LIN {X 0,Y 411.23,Z 342.072,A -85,B 0,C 180,E1 -10466.382,E2 -10466.382} C_VEL
LIN {X 0,Y 411.203,Z 342.077,A -85,B 0,C 180,E1 -10469.713,E2 -10469.713} C_VEL
LIN {X 0,Y 411.199,Z 342.079,A -85,B 0,C 180,E1 -10473.157,E2 -10473.157} C_VEL
LIN {X 0,Y 411.189,Z 342.079,A -85,B 0,C 180,E1 -10476.555,E2 -10476.555} C_VEL
LIN {X 0,Y 411.209,Z 342.075,A -85,B 0,C 180,E1 -10479.73,E2 -10479.73} C_VEL
LIN {X 0,Y 411.172,Z 342.082,A -85,B 0,C 180,E1 -10483.135,E2 -10483.135} C_VEL
LIN {X 0,Y 411.168,Z 342.08,A -85,B 0,C 180,E1 -10485.882,E2 -10485.882} C_VEL
LIN {X 0,Y 411.161,Z 342.084,A -85,B 0,C 180,E1 -10488.773,E2 -10488.773} C_VEL
LIN {X 0,Y 411.202,Z 342.076,A -85,B 0,C 180,E1 -10492.029,E2 -10492.029} C_VEL
LIN {X 0,Y 412.209,Z 347.522,A -85,B 0,C 180,E1 -10494.924,E2 -10494.924} C_VEL
LIN {X 0,Y 412.634,Z 351.681,A -85,B 0,C 180,E1 -10496.975,E2 -10496.975} C_VEL
LIN {X 0,Y 412.275,Z 356.532,A -85,B 0,C 180,E1 -10499.244,E2 -10499.244} C_VEL
LIN {X 0,Y 411.689,Z 363.91,A -85,B 0,C 180,E1 -10502.586,E2 -10502.586} C_VEL
LIN {X 0,Y 411.232,Z 371.157,A -85,B 0,C 180,E1 -10505.787,E2 -10505.787} C_VEL
LIN {X 0,Y 410.777,Z 379.693,A -85,B 0,C 180,E1 -10509.469,E2 -10509.469} C_VEL
LIN {X 0,Y 410.455,Z 388.245,A -85,B 0,C 180,E1 -10513.079,E2 -10513.079} C_VEL
LIN {X 0,Y 410.22,Z 395.922,A -85,B 0,C 180,E1 -10516.264,E2 -10516.264} C_VEL
LIN {X 0,Y 411.645,Z 408.983,A -85,B 0,C 180,E1 -10516.82,E2 -10516.82} C_VEL
LIN {X 0,Y 412.334,Z 417.705,A -85,B 0,C 180,E1 -10517.325,E2 -10517.325} C_VEL
LIN {X 0,Y 412.266,Z 426.417,A -85,B 0,C 180,E1 -10517.948,E2 -10517.948} C_VEL
LIN {X 0,Y 411.784,Z 434.733,A -85,B 0,C 180,E1 -10518.682,E2 -10518.682} C_VEL
LIN {X 0,Y 411.383,Z 442.624,A -85,B 0,C 180,E1 -10519.543,E2 -10519.543} C_VEL
LIN {X 0,Y 410.961,Z 449.152,A -85,B 0,C 180,E1 -10520.403,E2 -10520.403} C_VEL
LIN {X 0,Y 410.635,Z 455.373,A -85,B 0,C 180,E1 -10521.389,E2 -10521.389} C_VEL
LIN {X 0,Y 410.389,Z 460.538,A -85,B 0,C 180,E1 -10522.375,E2 -10522.375} C_VEL
LIN {X 0,Y 410.192,Z 464.991,A -85,B 0,C 180,E1 -10523.399,E2 -10523.399} C_VEL
LIN {X 0,Y 410.072,Z 469.17,A -85,B 0,C 180,E1 -10524.592,E2 -10524.592} C_VEL
LIN {X 0,Y 410.022,Z 471.91,A -85,B 0,C 180,E1 -10525.578,E2 -10525.578} C_VEL
LIN {X 0,Y 410.004,Z 474.894,A -85,B 0,C 180,E1 -10527.054,E2 -10527.054} C_VEL
LIN {X 0,Y 410.022,Z 476.211,A -85,B 0,C 180,E1 -10528.037,E2 -10528.037} C_VEL
LIN {X 0,Y 409.977,Z 477.041,A -85,B 0,C 180,E1 -10529.019,E2 -10529.019} C_VEL
LIN {X 0,Y 409.971,Z 477.337,A -85,B 0,C 180,E1 -10530.001,E2 -10530.001} C_VEL
LIN {X 0,Y 409.977,Z 477.054,A -85,B 0,C 180,E1 -10530.983,E2 -10530.983} C_VEL
LIN {X 0,Y 410.021,Z 476.298,A -85,B 0,C 180,E1 -10531.966,E2 -10531.966} C_VEL
LIN {X 0,Y 409.989,Z 475.058,A -85,B 0,C 180,E1 -10532.949,E2 -10532.949} C_VEL
LIN {X 0,Y 410.022,Z 472.138,A -85,B 0,C 180,E1 -10534.425,E2 -10534.425} C_VEL
LIN {X 0,Y 410.073,Z 469.497,A -85,B 0,C 180,E1 -10535.41,E2 -10535.41} C_VEL
LIN {X 0,Y 410.211,Z 465.349,A -85,B 0,C 180,E1 -10536.622,E2 -10536.622} C_VEL
LIN {X 0,Y 410.407,Z 461.101,A -85,B 0,C 180,E1 -10537.628,E2 -10537.628} C_VEL
LIN {X 0,Y 410.667,Z 456.097,A -85,B 0,C 180,E1 -10538.613,E2 -10538.613} C_VEL
LIN {X 0,Y 411.002,Z 450.082,A -85,B 0,C 180,E1 -10539.598,E2 -10539.598} C_VEL
LIN {X 0,Y 411.478,Z 442.783,A -85,B 0,C 180,E1 -10540.581,E2 -10540.581} C_VEL
LIN {X 0,Y 411.898,Z 435.006,A -85,B 0,C 180,E1 -10541.442,E2 -10541.442} C_VEL
LIN {X 0,Y 412.411,Z 426.855,A -85,B 0,C 180,E1 -10542.175,E2 -10542.175} C_VEL
LIN {X 0,Y 412.692,Z 420.277,A -85,B 0,C 180,E1 -10542.667,E2 -10542.667} C_VEL
LIN {X 0,Y 412.229,Z 412.315,A -85,B 0,C 180,E1 -10543.177,E2 -10543.177} C_VEL
LIN {X 0,Y 411.234,Z 402.961,A -85,B 0,C 180,E1 -10543.655,E2 -10543.655} C_VEL
LIN {X 0,Y 410.211,Z 395.094,A -85,B 0,C 180,E1 -10544.006,E2 -10544.006} C_VEL
LIN {X 0,Y 410.526,Z 386.814,A -85,B 0,C 180,E1 -10547.434,E2 -10547.434} C_VEL
LIN {X 0,Y 410.847,Z 378.285,A -85,B 0,C 180,E1 -10551.054,E2 -10551.054} C_VEL
LIN {X 0,Y 411.287,Z 370.025,A -85,B 0,C 180,E1 -10554.664,E2 -10554.664} C_VEL
LIN {X 0,Y 411.817,Z 362.717,A -85,B 0,C 180,E1 -10557.991,E2 -10557.991} C_VEL
LIN {X 0,Y 412.393,Z 356.864,A -85,B 0,C 180,E1 -10560.749,E2 -10560.749} C_VEL
LIN {X 0,Y 412.717,Z 352.266,A -85,B 0,C 180,E1 -10563.02,E2 -10563.02} C_VEL
LIN {X 0,Y 412.292,Z 348.349,A -85,B 0,C 180,E1 -10565.093,E2 -10565.093} C_VEL
LIN {X 0,Y 411.234,Z 342.076,A -85,B 0,C 180,E1 -10568.7,E2 -10568.7} C_VEL
LIN {X 0,Y 411.184,Z 342.088,A -85,B 0,C 180,E1 -10571.806,E2 -10571.806} C_VEL
LIN {X 0,Y 411.183,Z 342.084,A -85,B 0,C 180,E1 -10575.51,E2 -10575.51} C_VEL
LIN {X 0,Y 411.17,Z 342.083,A -85,B 0,C 180,E1 -10578.772,E2 -10578.772} C_VEL
LIN {X 0,Y 411.197,Z 342.079,A -85,B 0,C 180,E1 -10582.026,E2 -10582.026} C_VEL
LIN {X 0,Y 411.212,Z 342.078,A -85,B 0,C 180,E1 -10585.666,E2 -10585.666} C_VEL
LIN {X 0,Y 411.197,Z 342.079,A -85,B 0,C 180,E1 -10589.152,E2 -10589.152} C_VEL
LIN {X 0,Y 411.266,Z 342.069,A -85,B 0,C 180,E1 -10592.522,E2 -10592.522} C_VEL
LIN {X 0,Y 411.234,Z 342.074,A -85,B 0,C 180,E1 -10595.784,E2 -10595.784} C_VEL
LIN {X 0,Y 411.204,Z 342.079,A -85,B 0,C 180,E1 -10598.966,E2 -10598.966} C_VEL
LIN {X 0,Y 411.258,Z 342.071,A -85,B 0,C 180,E1 -10602.084,E2 -10602.084} C_VEL
LIN {X 0,Y 411.267,Z 342.07,A -85,B 0,C 180,E1 -10605.147,E2 -10605.147} C_VEL
LIN {X 0,Y 411.29,Z 342.068,A -85,B 0,C 180,E1 -10608.167,E2 -10608.167} C_VEL
LIN {X 0,Y 411.325,Z 342.062,A -85,B 0,C 180,E1 -10611.153,E2 -10611.153} C_VEL
LIN {X 0,Y 411.448,Z 342.048,A -85,B 0,C 180,E1 -10614.117,E2 -10614.117} C_VEL
LIN {X 0,Y 411.515,Z 342.037,A -85,B 0,C 180,E1 -10618.042,E2 -10618.042} C_VEL
LIN {X 0,Y 411.646,Z 342.024,A -85,B 0,C 180,E1 -10619.999,E2 -10619.999} C_VEL
LIN {X 0,Y 411.461,Z 342.045,A -85,B 0,C 180,E1 -10622.936,E2 -10622.936} C_VEL
LIN {X 0,Y 411.438,Z 342.048,A -85,B 0,C 180,E1 -10626.627,E2 -10626.627} C_VEL
LIN {X 0,Y 411.323,Z 342.062,A -85,B 0,C 180,E1 -10628.845,E2 -10628.845} C_VEL
LIN {X 0,Y 411.287,Z 342.069,A -85,B 0,C 180,E1 -10631.832,E2 -10631.832} C_VEL
LIN {X 0,Y 411.261,Z 342.074,A -85,B 0,C 180,E1 -10634.851,E2 -10634.851} C_VEL
LIN {X 0,Y 411.086,Z 342.096,A -85,B 0,C 180,E1 -10637.921,E2 -10637.921} C_VEL
LIN {X 0,Y 410.952,Z 342.111,A -85,B 0,C 180,E1 -10638.96,E2 -10638.96} C_VEL
LIN {X 0,Y 410.855,Z 342.735,A -85,B 0,C 180,E1 -10640.005,E2 -10640.005} C_VEL
LIN {X 0,Y 410.697,Z 346.204,A -85,B 0,C 180,E1 -10643.176,E2 -10643.176} C_VEL
LIN {X 0,Y 410.524,Z 349.853,A -85,B 0,C 180,E1 -10646.429,E2 -10646.429} C_VEL
LIN {X 0,Y 410.4,Z 353.677,A -85,B 0,C 180,E1 -10649.775,E2 -10649.775} C_VEL
LIN {X 0,Y 410.282,Z 357.723,A -85,B 0,C 180,E1 -10653.239,E2 -10653.239} C_VEL
LIN {X 0,Y 410.198,Z 361.362,A -85,B 0,C 180,E1 -10656.158,E2 -10656.158} C_VEL
LIN {X 0,Y 412.433,Z 371.958,A -85,B 0,C 180,E1 -10656.694,E2 -10656.694} C_VEL
LIN {X 0,Y 413.573,Z 378.962,A -85,B 0,C 180,E1 -10657.125,E2 -10657.125} C_VEL
LIN {X 0,Y 413.1,Z 389.049,A -85,B 0,C 180,E1 -10657.844,E2 -10657.844} C_VEL
LIN {X 0,Y 412.623,Z 397.601,A -85,B 0,C 180,E1 -10658.62,E2 -10658.62} C_VEL
LIN {X 0,Y 412.151,Z 405.235,A -85,B 0,C 180,E1 -10659.474,E2 -10659.474} C_VEL
LIN {X 0,Y 411.705,Z 412.313,A -85,B 0,C 180,E1 -10660.44,E2 -10660.44} C_VEL
LIN {X 0,Y 411.181,Z 420.303,A -85,B 0,C 180,E1 -10661.803,E2 -10661.803} C_VEL
LIN {X 0,Y 410.704,Z 426.486,A -85,B 0,C 180,E1 -10663.193,E2 -10663.193} C_VEL
LIN {X 0,Y 410.422,Z 431.277,A -85,B 0,C 180,E1 -10664.592,E2 -10664.592} C_VEL
LIN {X 0,Y 410.205,Z 434.884,A -85,B 0,C 180,E1 -10666.018,E2 -10666.018} C_VEL
LIN {X 0,Y 409.984,Z 437.361,A -85,B 0,C 180,E1 -10667.484,E2 -10667.484} C_VEL
LIN {X 0,Y 409.867,Z 438.729,A -85,B 0,C 180,E1 -10669.337,E2 -10669.337} C_VEL
LIN {X 0,Y 409.875,Z 438.684,A -85,B 0,C 180,E1 -10670.621,E2 -10670.621} C_VEL
LIN {X 0,Y 409.906,Z 437.633,A -85,B 0,C 180,E1 -10672.061,E2 -10672.061} C_VEL
LIN {X 0,Y 410.115,Z 435.241,A -85,B 0,C 180,E1 -10673.649,E2 -10673.649} C_VEL
LIN {X 0,Y 410.267,Z 432.368,A -85,B 0,C 180,E1 -10674.875,E2 -10674.875} C_VEL
LIN {X 0,Y 410.556,Z 427.036,A -85,B 0,C 180,E1 -10676.49,E2 -10676.49} C_VEL
LIN {X 0,Y 410.9,Z 421.655,A -85,B 0,C 180,E1 -10677.737,E2 -10677.737} C_VEL
LIN {X 0,Y 411.219,Z 416.518,A -85,B 0,C 180,E1 -10678.705,E2 -10678.705} C_VEL
LIN {X 0,Y 411.616,Z 409.786,A -85,B 0,C 180,E1 -10679.755,E2 -10679.755} C_VEL
LIN {X 0,Y 411.963,Z 402.423,A -85,B 0,C 180,E1 -10680.698,E2 -10680.698} C_VEL
LIN {X 0,Y 412.553,Z 392.414,A -85,B 0,C 180,E1 -10681.717,E2 -10681.717} C_VEL
LIN {X 0,Y 412.981,Z 382.762,A -85,B 0,C 180,E1 -10682.465,E2 -10682.465} C_VEL
LIN {X 0,Y 413.008,Z 376.343,A -85,B 0,C 180,E1 -10682.88,E2 -10682.88} C_VEL
LIN {X 0,Y 411.176,Z 365.69,A -85,B 0,C 180,E1 -10683.452,E2 -10683.452} C_VEL
LIN {X 0,Y 410.147,Z 360.352,A -85,B 0,C 180,E1 -10683.714,E2 -10683.714} C_VEL
LIN {X 0,Y 410.174,Z 356.533,A -85,B 0,C 180,E1 -10686.79,E2 -10686.79} C_VEL
LIN {X 0,Y 410.288,Z 352.106,A -85,B 0,C 180,E1 -10690.406,E2 -10690.406} C_VEL
LIN {X 0,Y 410.442,Z 348.369,A -85,B 0,C 180,E1 -10693.508,E2 -10693.508} C_VEL
LIN {X 0,Y 410.61,Z 343.854,A -85,B 0,C 180,E1 -10697.313,E2 -10697.313} C_VEL
LIN {X 0,Y 410.673,Z 342.882,A -85,B 0,C 180,E1 -10698.148,E2 -10698.148} C_VEL
LIN {X 0,Y 410.706,Z 342.14,A -85,B 0,C 180,E1 -10699.149,E2 -10699.149} C_VEL
LIN {X 0,Y 411.303,Z 342.067,A -85,B 0,C 180,E1 -10702.319,E2 -10702.319} C_VEL
LIN {X 0,Y 411.449,Z 342.048,A -85,B 0,C 180,E1 -10704.116,E2 -10704.116} C_VEL
LIN {X 0,Y 411.504,Z 342.041,A -85,B 0,C 180,E1 -10708.041,E2 -10708.041} C_VEL
LIN {X 0,Y 411.631,Z 342.025,A -85,B 0,C 180,E1 -10709.999,E2 -10709.999} C_VEL
LIN {X 0,Y 411.457,Z 342.044,A -85,B 0,C 180,E1 -10712.936,E2 -10712.936} C_VEL
LIN {X 0,Y 411.482,Z 342.045,A -85,B 0,C 180,E1 -10715.881,E2 -10715.881} C_VEL
LIN {X 0,Y 411.444,Z 342.045,A -85,B 0,C 180,E1 -10717.13,E2 -10717.13} C_VEL
LIN {X 0,Y 410.763,Z 342.134,A -85,B 0,C 180,E1 -10717.947,E2 -10717.947} C_VEL
LIN {X 0,Y 407.846,Z 342.494,A -85,B 0,C 180,E1 -10719.272,E2 -10719.272} C_VEL
LIN {X 0,Y 405.379,Z 342.803,A -85,B 0,C 180,E1 -10720.343,E2 -10720.343} C_VEL
LIN {X 0,Y 404.323,Z 342.933,A -85,B 0,C 180,E1 -10721.172,E2 -10721.172} C_VEL
LIN {X 0,Y 404.239,Z 342.942,A -85,B 0,C 180,E1 -10721.452,E2 -10721.452} C_VEL
LIN {X 0,Y 404.204,Z 342.95,A -85,B 0,C 180,E1 -10724.087,E2 -10724.087} C_VEL
LIN {X 0,Y 404.19,Z 342.951,A -85,B 0,C 180,E1 -10727.192,E2 -10727.192} C_VEL
LIN {X 0,Y 404.15,Z 342.954,A -85,B 0,C 180,E1 -10730.351,E2 -10730.351} C_VEL
LIN {X 0,Y 404.156,Z 342.957,A -85,B 0,C 180,E1 -10733.574,E2 -10733.574} C_VEL
LIN {X 0,Y 404.17,Z 342.954,A -85,B 0,C 180,E1 -10735.766,E2 -10735.766} C_VEL
LIN {X 0,Y 404.184,Z 342.951,A -85,B 0,C 180,E1 -10737.999,E2 -10737.999} C_VEL
LIN {X 0,Y 404.129,Z 342.959,A -85,B 0,C 180,E1 -10741.558,E2 -10741.558} C_VEL
LIN {X 0,Y 404.171,Z 342.954,A -85,B 0,C 180,E1 -10745.016,E2 -10745.016} C_VEL
LIN {X 0,Y 404.149,Z 342.956,A -85,B 0,C 180,E1 -10748.755,E2 -10748.755} C_VEL
LIN {X 0,Y 404.177,Z 342.953,A -85,B 0,C 180,E1 -10751.61,E2 -10751.61} C_VEL
LIN {X 0,Y 404.184,Z 342.951,A -85,B 0,C 180,E1 -10754.53,E2 -10754.53} C_VEL
LIN {X 0,Y 404.192,Z 342.951,A -85,B 0,C 180,E1 -10757.305,E2 -10757.305} C_VEL
LIN {X 0,Y 404.154,Z 342.953,A -85,B 0,C 180,E1 -10759.955,E2 -10759.955} C_VEL
LIN {X 0,Y 404.126,Z 342.959,A -85,B 0,C 180,E1 -10763.124,E2 -10763.124} C_VEL
LIN {X 0,Y 404.13,Z 342.957,A -85,B 0,C 180,E1 -10766.188,E2 -10766.188} C_VEL
LIN {X 0,Y 404.14,Z 342.954,A -85,B 0,C 180,E1 -10769.716,E2 -10769.716} C_VEL
LIN {X 0,Y 404.181,Z 342.951,A -85,B 0,C 180,E1 -10773.123,E2 -10773.123} C_VEL
LIN {X 0,Y 404.169,Z 342.955,A -85,B 0,C 180,E1 -10776.427,E2 -10776.427} C_VEL
LIN {X 0,Y 404.213,Z 342.946,A -85,B 0,C 180,E1 -10779.861,E2 -10779.861} C_VEL
LIN {X 0,Y 404.205,Z 342.948,A -85,B 0,C 180,E1 -10782.992,E2 -10782.992} C_VEL
LIN {X 0,Y 404.253,Z 342.943,A -85,B 0,C 180,E1 -10786.789,E2 -10786.789} C_VEL
LIN {X 0,Y 404.258,Z 342.944,A -85,B 0,C 180,E1 -10789.989,E2 -10789.989} C_VEL
LIN {X 0,Y 404.4,Z 342.923,A -85,B 0,C 180,E1 -10793.014,E2 -10793.014} C_VEL
LIN {X 0,Y 404.273,Z 342.938,A -85,B 0,C 180,E1 -10795.015,E2 -10795.015} C_VEL
LIN {X 0,Y 404.471,Z 342.917,A -85,B 0,C 180,E1 -10798.009,E2 -10798.009} C_VEL
LIN {X 0,Y 404.6,Z 342.901,A -85,B 0,C 180,E1 -10800.001,E2 -10800.001} C_VEL
LIN {X 0,Y 404.415,Z 342.921,A -85,B 0,C 180,E1 -10802.989,E2 -10802.989} C_VEL
LIN {X 0,Y 404.401,Z 342.923,A -85,B 0,C 180,E1 -10806.988,E2 -10806.988} C_VEL
LIN {X 0,Y 404.261,Z 342.943,A -85,B 0,C 180,E1 -10810.013,E2 -10810.013} C_VEL
LIN {X 0,Y 404.256,Z 342.943,A -85,B 0,C 180,E1 -10813.213,E2 -10813.213} C_VEL
LIN {X 0,Y 404.206,Z 342.949,A -85,B 0,C 180,E1 -10817.008,E2 -10817.008} C_VEL
LIN {X 0,Y 404.155,Z 342.953,A -85,B 0,C 180,E1 -10820.353,E2 -10820.353} C_VEL
LIN {X 0,Y 404.161,Z 342.956,A -85,B 0,C 180,E1 -10823.576,E2 -10823.576} C_VEL
LIN {X 0,Y 404.175,Z 342.953,A -85,B 0,C 180,E1 -10825.768,E2 -10825.768} C_VEL
LIN {X 0,Y 404.19,Z 342.949,A -85,B 0,C 180,E1 -10828.001,E2 -10828.001} C_VEL
LIN {X 0,Y 404.135,Z 342.958,A -85,B 0,C 180,E1 -10831.56,E2 -10831.56} C_VEL
LIN {X 0,Y 404.178,Z 342.954,A -85,B 0,C 180,E1 -10835.017,E2 -10835.017} C_VEL
LIN {X 0,Y 404.151,Z 342.957,A -85,B 0,C 180,E1 -10838.758,E2 -10838.758} C_VEL
LIN {X 0,Y 404.118,Z 342.959,A -85,B 0,C 180,E1 -10841.601,E2 -10841.601} C_VEL
LIN {X 0,Y 404.144,Z 342.957,A -85,B 0,C 180,E1 -10844.524,E2 -10844.524} C_VEL
LIN {X 0,Y 404.134,Z 342.958,A -85,B 0,C 180,E1 -10847.298,E2 -10847.298} C_VEL
LIN {X 0,Y 404.164,Z 342.954,A -85,B 0,C 180,E1 -10849.957,E2 -10849.957} C_VEL
LIN {X 0,Y 404.201,Z 343.069,A -85,B 0,C 180,E1 -10851.965,E2 -10851.965} C_VEL
LIN {X 0,Y 405.47,Z 350.234,A -85,B 0,C 180,E1 -10855.717,E2 -10855.717} C_VEL
LIN {X 0,Y 405.604,Z 353.875,A -85,B 0,C 180,E1 -10857.512,E2 -10857.512} C_VEL
LIN {X 0,Y 404.93,Z 361.148,A -85,B 0,C 180,E1 -10860.926,E2 -10860.926} C_VEL
LIN {X 0,Y 404.403,Z 368.438,A -85,B 0,C 180,E1 -10864.25,E2 -10864.25} C_VEL
LIN {X 0,Y 403.922,Z 375.737,A -85,B 0,C 180,E1 -10867.495,E2 -10867.495} C_VEL
LIN {X 0,Y 403.561,Z 383.066,A -85,B 0,C 180,E1 -10870.679,E2 -10870.679} C_VEL
LIN {X 0,Y 403.312,Z 390.352,A -85,B 0,C 180,E1 -10873.812,E2 -10873.812} C_VEL
LIN {X 0,Y 403.117,Z 395.66,A -85,B 0,C 180,E1 -10876.058,E2 -10876.058} C_VEL
LIN {X 0,Y 404.579,Z 408.507,A -85,B 0,C 180,E1 -10876.603,E2 -10876.603} C_VEL
LIN {X 0,Y 405.268,Z 417.013,A -85,B 0,C 180,E1 -10877.1,E2 -10877.1} C_VEL
LIN {X 0,Y 405.302,Z 425.811,A -85,B 0,C 180,E1 -10877.737,E2 -10877.737} C_VEL
LIN {X 0,Y 404.817,Z 434.179,A -85,B 0,C 180,E1 -10878.485,E2 -10878.485} C_VEL
LIN {X 0,Y 404.396,Z 442.112,A -85,B 0,C 180,E1 -10879.361,E2 -10879.361} C_VEL
LIN {X 0,Y 403.94,Z 448.67,A -85,B 0,C 180,E1 -10880.235,E2 -10880.235} C_VEL
LIN {X 0,Y 403.601,Z 454.919,A -85,B 0,C 180,E1 -10881.237,E2 -10881.237} C_VEL
LIN {X 0,Y 403.327,Z 460.107,A -85,B 0,C 180,E1 -10882.24,E2 -10882.24} C_VEL
LIN {X 0,Y 403.116,Z 464.859,A -85,B 0,C 180,E1 -10883.356,E2 -10883.356} C_VEL
LIN {X 0,Y 402.972,Z 468.776,A -85,B 0,C 180,E1 -10884.497,E2 -10884.497} C_VEL
LIN {X 0,Y 402.952,Z 471.534,A -85,B 0,C 180,E1 -10885.5,E2 -10885.5} C_VEL
LIN {X 0,Y 402.904,Z 474.529,A -85,B 0,C 180,E1 -10887.002,E2 -10887.002} C_VEL
LIN {X 0,Y 402.951,Z 475.861,A -85,B 0,C 180,E1 -10888.002,E2 -10888.002} C_VEL
LIN {X 0,Y 402.902,Z 476.702,A -85,B 0,C 180,E1 -10889.002,E2 -10889.002} C_VEL
LIN {X 0,Y 402.894,Z 477,A -85,B 0,C 180,E1 -10890.001,E2 -10890.001} C_VEL
LIN {X 0,Y 402.902,Z 476.726,A -85,B 0,C 180,E1 -10891.001,E2 -10891.001} C_VEL
LIN {X 0,Y 402.95,Z 475.982,A -85,B 0,C 180,E1 -10892,E2 -10892} C_VEL
LIN {X 0,Y 402.888,Z 474.753,A -85,B 0,C 180,E1 -10893.001,E2 -10893.001} C_VEL
LIN {X 0,Y 402.952,Z 471.848,A -85,B 0,C 180,E1 -10894.503,E2 -10894.503} C_VEL
LIN {X 0,Y 402.971,Z 469.219,A -85,B 0,C 180,E1 -10895.506,E2 -10895.506} C_VEL
LIN {X 0,Y 403.137,Z 465.344,A -85,B 0,C 180,E1 -10896.672,E2 -10896.672} C_VEL
LIN {X 0,Y 403.359,Z 460.853,A -85,B 0,C 180,E1 -10897.762,E2 -10897.762} C_VEL
LIN {X 0,Y 403.617,Z 455.866,A -85,B 0,C 180,E1 -10898.765,E2 -10898.765} C_VEL
LIN {X 0,Y 403.988,Z 449.872,A -85,B 0,C 180,E1 -10899.767,E2 -10899.767} C_VEL
LIN {X 0,Y 404.5,Z 442.599,A -85,B 0,C 180,E1 -10900.766,E2 -10900.766} C_VEL
LIN {X 0,Y 404.947,Z 434.855,A -85,B 0,C 180,E1 -10901.641,E2 -10901.641} C_VEL
LIN {X 0,Y 405.48,Z 426.747,A -85,B 0,C 180,E1 -10902.387,E2 -10902.387} C_VEL
LIN {X 0,Y 405.686,Z 420.228,A -85,B 0,C 180,E1 -10902.889,E2 -10902.889} C_VEL
LIN {X 0,Y 405.115,Z 411.093,A -85,B 0,C 180,E1 -10903.481,E2 -10903.481} C_VEL
LIN {X 0,Y 404.054,Z 401.482,A -85,B 0,C 180,E1 -10903.97,E2 -10903.97} C_VEL
LIN {X 0,Y 403.148,Z 394.806,A -85,B 0,C 180,E1 -10904.256,E2 -10904.256} C_VEL
LIN {X 0,Y 403.457,Z 386.563,A -85,B 0,C 180,E1 -10907.75,E2 -10907.75} C_VEL
LIN {X 0,Y 403.81,Z 378.069,A -85,B 0,C 180,E1 -10911.439,E2 -10911.439} C_VEL
LIN {X 0,Y 404.239,Z 370.846,A -85,B 0,C 180,E1 -10914.663,E2 -10914.663} C_VEL
LIN {X 0,Y 404.786,Z 363.737,A -85,B 0,C 180,E1 -10917.956,E2 -10917.956} C_VEL
LIN {X 0,Y 405.441,Z 356.773,A -85,B 0,C 180,E1 -10921.335,E2 -10921.335} C_VEL
LIN {X 0,Y 405.723,Z 353.363,A -85,B 0,C 180,E1 -10923.07,E2 -10923.07} C_VEL
LIN {X 0,Y 405.359,Z 349.966,A -85,B 0,C 180,E1 -10924.901,E2 -10924.901} C_VEL
LIN {X 0,Y 404.324,Z 343.717,A -85,B 0,C 180,E1 -10928.537,E2 -10928.537} C_VEL
LIN {X 0,Y 404.185,Z 342.955,A -85,B 0,C 180,E1 -10929.075,E2 -10929.075} C_VEL
LIN {X 0,Y 404.16,Z 342.963,A -85,B 0,C 180,E1 -10933.084,E2 -10933.084} C_VEL
LIN {X 0,Y 404.155,Z 342.959,A -85,B 0,C 180,E1 -10935.926,E2 -10935.926} C_VEL
LIN {X 0,Y 404.125,Z 342.961,A -85,B 0,C 180,E1 -10938.635,E2 -10938.635} C_VEL
LIN {X 0,Y 404.155,Z 342.956,A -85,B 0,C 180,E1 -10941.493,E2 -10941.493} C_VEL
LIN {X 0,Y 404.191,Z 342.952,A -85,B 0,C 180,E1 -10944.984,E2 -10944.984} C_VEL
LIN {X 0,Y 404.149,Z 342.957,A -85,B 0,C 180,E1 -10948.554,E2 -10948.554} C_VEL
LIN {X 0,Y 404.203,Z 342.95,A -85,B 0,C 180,E1 -10952,E2 -10952} C_VEL
LIN {X 0,Y 404.185,Z 342.953,A -85,B 0,C 180,E1 -10955.334,E2 -10955.334} C_VEL
LIN {X 0,Y 404.146,Z 342.957,A -85,B 0,C 180,E1 -10958.58,E2 -10958.58} C_VEL
LIN {X 0,Y 404.216,Z 342.947,A -85,B 0,C 180,E1 -10961.761,E2 -10961.761} C_VEL
LIN {X 0,Y 404.213,Z 342.95,A -85,B 0,C 180,E1 -10964.881,E2 -10964.881} C_VEL
LIN {X 0,Y 404.262,Z 342.942,A -85,B 0,C 180,E1 -10967.958,E2 -10967.958} C_VEL
LIN {X 0,Y 404.272,Z 342.941,A -85,B 0,C 180,E1 -10970.998,E2 -10970.998} C_VEL
LIN {X 0,Y 404.398,Z 342.926,A -85,B 0,C 180,E1 -10974.014,E2 -10974.014} C_VEL
LIN {X 0,Y 404.484,Z 342.913,A -85,B 0,C 180,E1 -10978.008,E2 -10978.008} C_VEL
LIN {X 0,Y 404.615,Z 342.9,A -85,B 0,C 180,E1 -10979.999,E2 -10979.999} C_VEL
LIN {X 0,Y 404.419,Z 342.922,A -85,B 0,C 180,E1 -10982.987,E2 -10982.987} C_VEL
LIN {X 0,Y 404.387,Z 342.926,A -85,B 0,C 180,E1 -10986.625,E2 -10986.625} C_VEL
LIN {X 0,Y 404.261,Z 342.943,A -85,B 0,C 180,E1 -10990.011,E2 -10990.011} C_VEL
LIN {X 0,Y 404.271,Z 342.945,A -85,B 0,C 180,E1 -10993.21,E2 -10993.21} C_VEL
LIN {X 0,Y 404.204,Z 342.954,A -85,B 0,C 180,E1 -10996.151,E2 -10996.151} C_VEL
LIN {X 0,Y 403.844,Z 342.997,A -85,B 0,C 180,E1 -10999.307,E2 -10999.307} C_VEL
LIN {X 0,Y 403.694,Z 346.515,A -85,B 0,C 180,E1 -11002.676,E2 -11002.676} C_VEL
LIN {X 0,Y 403.5,Z 350.007,A -85,B 0,C 180,E1 -11005.812,E2 -11005.812} C_VEL
LIN {X 0,Y 403.359,Z 354.027,A -85,B 0,C 180,E1 -11009.402,E2 -11009.402} C_VEL
LIN {X 0,Y 403.229,Z 357.821,A -85,B 0,C 180,E1 -11012.703,E2 -11012.703} C_VEL
LIN {X 0,Y 403.109,Z 361.529,A -85,B 0,C 180,E1 -11015.869,E2 -11015.869} C_VEL
LIN {X 0,Y 405.442,Z 372.434,A -85,B 0,C 180,E1 -11016.443,E2 -11016.443} C_VEL
LIN {X 0,Y 406.673,Z 379.898,A -85,B 0,C 180,E1 -11016.923,E2 -11016.923} C_VEL
LIN {X 0,Y 406.245,Z 388.915,A -85,B 0,C 180,E1 -11017.574,E2 -11017.574} C_VEL
LIN {X 0,Y 405.797,Z 396.48,A -85,B 0,C 180,E1 -11018.252,E2 -11018.252} C_VEL
LIN {X 0,Y 405.348,Z 403.228,A -85,B 0,C 180,E1 -11018.979,E2 -11018.979} C_VEL
LIN {X 0,Y 404.874,Z 410.673,A -85,B 0,C 180,E1 -11019.959,E2 -11019.959} C_VEL
LIN {X 0,Y 404.441,Z 417.301,A -85,B 0,C 180,E1 -11021.026,E2 -11021.026} C_VEL
LIN {X 0,Y 404.106,Z 421.562,A -85,B 0,C 180,E1 -11021.836,E2 -11021.836} C_VEL
LIN {X 0,Y 403.686,Z 426.671,A -85,B 0,C 180,E1 -11023.012,E2 -11023.012} C_VEL
LIN {X 0,Y 403.436,Z 430.702,A -85,B 0,C 180,E1 -11024.17,E2 -11024.17} C_VEL
LIN {X 0,Y 403.183,Z 434.518,A -85,B 0,C 180,E1 -11025.615,E2 -11025.615} C_VEL
LIN {X 0,Y 402.936,Z 437.29,A -85,B 0,C 180,E1 -11027.137,E2 -11027.137} C_VEL
LIN {X 0,Y 402.828,Z 438.814,A -85,B 0,C 180,E1 -11028.606,E2 -11028.606} C_VEL
LIN {X 0,Y 402.761,Z 439.179,A -85,B 0,C 180,E1 -11030.153,E2 -11030.153} C_VEL
LIN {X 0,Y 402.799,Z 438.304,A -85,B 0,C 180,E1 -11031.733,E2 -11031.733} C_VEL
LIN {X 0,Y 402.847,Z 437.676,A -85,B 0,C 180,E1 -11032.366,E2 -11032.366} C_VEL
LIN {X 0,Y 403.025,Z 435.668,A -85,B 0,C 180,E1 -11033.636,E2 -11033.636} C_VEL
LIN {X 0,Y 403.194,Z 432.506,A -85,B 0,C 180,E1 -11035.007,E2 -11035.007} C_VEL
LIN {X 0,Y 403.461,Z 427.845,A -85,B 0,C 180,E1 -11036.454,E2 -11036.454} C_VEL
LIN {X 0,Y 403.802,Z 422.952,A -85,B 0,C 180,E1 -11037.641,E2 -11037.641} C_VEL
LIN {X 0,Y 404.054,Z 418.484,A -85,B 0,C 180,E1 -11038.545,E2 -11038.545} C_VEL
LIN {X 0,Y 404.537,Z 411.162,A -85,B 0,C 180,E1 -11039.746,E2 -11039.746} C_VEL
LIN {X 0,Y 404.925,Z 404.086,A -85,B 0,C 180,E1 -11040.694,E2 -11040.694} C_VEL
LIN {X 0,Y 405.364,Z 396.557,A -85,B 0,C 180,E1 -11041.524,E2 -11041.524} C_VEL
LIN {X 0,Y 405.858,Z 386.656,A -85,B 0,C 180,E1 -11042.404,E2 -11042.404} C_VEL
LIN {X 0,Y 406.177,Z 378.2,A -85,B 0,C 180,E1 -11042.985,E2 -11042.985} C_VEL
LIN {X 0,Y 404.21,Z 366.469,A -85,B 0,C 180,E1 -11043.645,E2 -11043.645} C_VEL
LIN {X 0,Y 403.075,Z 360.681,A -85,B 0,C 180,E1 -11043.913,E2 -11043.913} C_VEL
LIN {X 0,Y 403.098,Z 357.669,A -85,B 0,C 180,E1 -11046.358,E2 -11046.358} C_VEL
LIN {X 0,Y 403.213,Z 352.945,A -85,B 0,C 180,E1 -11050.252,E2 -11050.252} C_VEL
LIN {X 0,Y 403.383,Z 348.711,A -85,B 0,C 180,E1 -11053.812,E2 -11053.812} C_VEL
LIN {X 0,Y 403.541,Z 344.704,A -85,B 0,C 180,E1 -11057.228,E2 -11057.228} C_VEL
LIN {X 0,Y 403.628,Z 343.023,A -85,B 0,C 180,E1 -11058.957,E2 -11058.957} C_VEL
LIN {X 0,Y 404.246,Z 342.946,A -85,B 0,C 180,E1 -11062.283,E2 -11062.283} C_VEL
LIN {X 0,Y 404.391,Z 342.927,A -85,B 0,C 180,E1 -11064.013,E2 -11064.013} C_VEL
LIN {X 0,Y 404.473,Z 342.917,A -85,B 0,C 180,E1 -11068.007,E2 -11068.007} C_VEL
LIN {X 0,Y 404.601,Z 342.901,A -85,B 0,C 180,E1 -11069.999,E2 -11069.999} C_VEL
LIN {X 0,Y 404.414,Z 342.921,A -85,B 0,C 180,E1 -11072.987,E2 -11072.987} C_VEL
LIN {X 0,Y 404.428,Z 342.923,A -85,B 0,C 180,E1 -11075.984,E2 -11075.984} C_VEL
LIN {X 0,Y 404.411,Z 342.925,A -85,B 0,C 180,E1 -11077.99,E2 -11077.99} C_VEL
LIN {X 0,Y 404.239,Z 342.942,A -85,B 0,C 180,E1 -11081.452,E2 -11081.452} C_VEL
LIN {X 0,Y 403.574,Z 343.028,A -85,B 0,C 180,E1 -11082.284,E2 -11082.284} C_VEL
LIN {X 0,Y 400.709,Z 343.385,A -85,B 0,C 180,E1 -11083.636,E2 -11083.636} C_VEL
LIN {X 0,Y 398.279,Z 343.687,A -85,B 0,C 180,E1 -11084.728,E2 -11084.728} C_VEL
LIN {X 0,Y 397.232,Z 343.819,A -85,B 0,C 180,E1 -11085.573,E2 -11085.573} C_VEL
LIN {X 0,Y 397.145,Z 343.826,A -85,B 0,C 180,E1 -11085.859,E2 -11085.859} C_VEL
LIN {X 0,Y 397.149,Z 343.826,A -85,B 0,C 180,E1 -11088.573,E2 -11088.573} C_VEL
LIN {X 0,Y 397.083,Z 343.837,A -85,B 0,C 180,E1 -11091.818,E2 -11091.818} C_VEL
LIN {X 0,Y 397.143,Z 343.828,A -85,B 0,C 180,E1 -11095.131,E2 -11095.131} C_VEL
LIN {X 0,Y 397.149,Z 343.828,A -85,B 0,C 180,E1 -11097.776,E2 -11097.776} C_VEL
LIN {X 0,Y 397.07,Z 343.837,A -85,B 0,C 180,E1 -11100.881,E2 -11100.881} C_VEL
LIN {X 0,Y 397.111,Z 343.83,A -85,B 0,C 180,E1 -11104.493,E2 -11104.493} C_VEL
LIN {X 0,Y 397.096,Z 343.832,A -85,B 0,C 180,E1 -11108.274,E2 -11108.274} C_VEL
LIN {X 0,Y 397.141,Z 343.827,A -85,B 0,C 180,E1 -11111.993,E2 -11111.993} C_VEL
LIN {X 0,Y 397.135,Z 343.831,A -85,B 0,C 180,E1 -11115.06,E2 -11115.06} C_VEL
LIN {X 0,Y 397.141,Z 343.827,A -85,B 0,C 180,E1 -11118.007,E2 -11118.007} C_VEL
LIN {X 0,Y 397.096,Z 343.833,A -85,B 0,C 180,E1 -11121.726,E2 -11121.726} C_VEL
LIN {X 0,Y 397.111,Z 343.831,A -85,B 0,C 180,E1 -11125.507,E2 -11125.507} C_VEL
LIN {X 0,Y 397.072,Z 343.837,A -85,B 0,C 180,E1 -11129.119,E2 -11129.119} C_VEL
LIN {X 0,Y 397.18,Z 343.826,A -85,B 0,C 180,E1 -11132.61,E2 -11132.61} C_VEL
LIN {X 0,Y 397.126,Z 343.83,A -85,B 0,C 180,E1 -11135.983,E2 -11135.983} C_VEL
LIN {X 0,Y 397.143,Z 343.826,A -85,B 0,C 180,E1 -11139.274,E2 -11139.274} C_VEL
LIN {X 0,Y 397.17,Z 343.825,A -85,B 0,C 180,E1 -11142.844,E2 -11142.844} C_VEL
LIN {X 0,Y 397.17,Z 343.824,A -85,B 0,C 180,E1 -11145.658,E2 -11145.658} C_VEL
LIN {X 0,Y 397.197,Z 343.82,A -85,B 0,C 180,E1 -11148.778,E2 -11148.778} C_VEL
LIN {X 0,Y 397.382,Z 343.8,A -85,B 0,C 180,E1 -11152.042,E2 -11152.042} C_VEL
LIN {X 0,Y 397.244,Z 343.813,A -85,B 0,C 180,E1 -11154.926,E2 -11154.926} C_VEL
LIN {X 0,Y 397.44,Z 343.793,A -85,B 0,C 180,E1 -11157.974,E2 -11157.974} C_VEL
LIN {X 0,Y 397.569,Z 343.777,A -85,B 0,C 180,E1 -11160.001,E2 -11160.001} C_VEL
LIN {X 0,Y 397.373,Z 343.798,A -85,B 0,C 180,E1 -11163.042,E2 -11163.042} C_VEL
LIN {X 0,Y 397.353,Z 343.801,A -85,B 0,C 180,E1 -11167.113,E2 -11167.113} C_VEL
LIN {X 0,Y 397.219,Z 343.819,A -85,B 0,C 180,E1 -11170.192,E2 -11170.192} C_VEL
LIN {X 0,Y 397.217,Z 343.821,A -85,B 0,C 180,E1 -11173.322,E2 -11173.322} C_VEL
LIN {X 0,Y 397.172,Z 343.825,A -85,B 0,C 180,E1 -11177.156,E2 -11177.156} C_VEL
LIN {X 0,Y 397.094,Z 343.833,A -85,B 0,C 180,E1 -11180.731,E2 -11180.731} C_VEL
LIN {X 0,Y 397.124,Z 343.829,A -85,B 0,C 180,E1 -11184.02,E2 -11184.02} C_VEL
LIN {X 0,Y 397.187,Z 343.825,A -85,B 0,C 180,E1 -11187.391,E2 -11187.391} C_VEL
LIN {X 0,Y 397.077,Z 343.837,A -85,B 0,C 180,E1 -11190.883,E2 -11190.883} C_VEL
LIN {X 0,Y 397.119,Z 343.83,A -85,B 0,C 180,E1 -11194.495,E2 -11194.495} C_VEL
LIN {X 0,Y 397.099,Z 343.832,A -85,B 0,C 180,E1 -11198.276,E2 -11198.276} C_VEL
LIN {X 0,Y 397.083,Z 343.838,A -85,B 0,C 180,E1 -11200.91,E2 -11200.91} C_VEL
LIN {X 0,Y 397.098,Z 343.832,A -85,B 0,C 180,E1 -11203.65,E2 -11203.65} C_VEL
LIN {X 0,Y 397.1,Z 343.834,A -85,B 0,C 180,E1 -11206.522,E2 -11206.522} C_VEL
LIN {X 0,Y 397.111,Z 343.833,A -85,B 0,C 180,E1 -11210.425,E2 -11210.425} C_VEL
LIN {X 0,Y 397.142,Z 343.893,A -85,B 0,C 180,E1 -11211.732,E2 -11211.732} C_VEL
LIN {X 0,Y 398.238,Z 349.993,A -85,B 0,C 180,E1 -11215.004,E2 -11215.004} C_VEL
LIN {X 0,Y 398.604,Z 353.628,A -85,B 0,C 180,E1 -11216.869,E2 -11216.869} C_VEL
LIN {X 0,Y 398.097,Z 359.888,A -85,B 0,C 180,E1 -11219.889,E2 -11219.889} C_VEL
LIN {X 0,Y 397.507,Z 366.949,A -85,B 0,C 180,E1 -11223.204,E2 -11223.204} C_VEL
LIN {X 0,Y 397,Z 374.243,A -85,B 0,C 180,E1 -11226.53,E2 -11226.53} C_VEL
LIN {X 0,Y 396.576,Z 381.837,A -85,B 0,C 180,E1 -11229.927,E2 -11229.927} C_VEL
LIN {X 0,Y 396.245,Z 390.015,A -85,B 0,C 180,E1 -11233.515,E2 -11233.515} C_VEL
LIN {X 0,Y 396.049,Z 395.374,A -85,B 0,C 180,E1 -11235.833,E2 -11235.833} C_VEL
LIN {X 0,Y 397.489,Z 407.945,A -85,B 0,C 180,E1 -11236.373,E2 -11236.373} C_VEL
LIN {X 0,Y 398.291,Z 418.186,A -85,B 0,C 180,E1 -11237,E2 -11237} C_VEL
LIN {X 0,Y 398.341,Z 425.189,A -85,B 0,C 180,E1 -11237.52,E2 -11237.52} C_VEL
LIN {X 0,Y 397.82,Z 433.607,A -85,B 0,C 180,E1 -11238.28,E2 -11238.28} C_VEL
LIN {X 0,Y 397.373,Z 441.579,A -85,B 0,C 180,E1 -11239.17,E2 -11239.17} C_VEL
LIN {X 0,Y 396.93,Z 448.173,A -85,B 0,C 180,E1 -11240.061,E2 -11240.061} C_VEL
LIN {X 0,Y 396.572,Z 454.45,A -85,B 0,C 180,E1 -11241.081,E2 -11241.081} C_VEL
LIN {X 0,Y 396.273,Z 459.662,A -85,B 0,C 180,E1 -11242.101,E2 -11242.101} C_VEL
LIN {X 0,Y 396.022,Z 464.968,A -85,B 0,C 180,E1 -11243.378,E2 -11243.378} C_VEL
LIN {X 0,Y 395.874,Z 468.37,A -85,B 0,C 180,E1 -11244.398,E2 -11244.398} C_VEL
LIN {X 0,Y 395.881,Z 471.148,A -85,B 0,C 180,E1 -11245.419,E2 -11245.419} C_VEL
LIN {X 0,Y 395.805,Z 474.159,A -85,B 0,C 180,E1 -11246.948,E2 -11246.948} C_VEL
LIN {X 0,Y 395.881,Z 475.507,A -85,B 0,C 180,E1 -11247.967,E2 -11247.967} C_VEL
LIN {X 0,Y 395.83,Z 476.362,A -85,B 0,C 180,E1 -11248.984,E2 -11248.984} C_VEL
LIN {X 0,Y 395.819,Z 476.66,A -85,B 0,C 180,E1 -11250.001,E2 -11250.001} C_VEL
LIN {X 0,Y 395.83,Z 476.398,A -85,B 0,C 180,E1 -11251.019,E2 -11251.019} C_VEL
LIN {X 0,Y 395.861,Z 475.667,A -85,B 0,C 180,E1 -11252.036,E2 -11252.036} C_VEL
LIN {X 0,Y 395.788,Z 474.45,A -85,B 0,C 180,E1 -11253.055,E2 -11253.055} C_VEL
LIN {X 0,Y 395.882,Z 471.558,A -85,B 0,C 180,E1 -11254.583,E2 -11254.583} C_VEL
LIN {X 0,Y 395.912,Z 467.389,A -85,B 0,C 180,E1 -11256.115,E2 -11256.115} C_VEL
LIN {X 0,Y 396.242,Z 461.776,A -85,B 0,C 180,E1 -11257.646,E2 -11257.646} C_VEL
LIN {X 0,Y 396.582,Z 455.636,A -85,B 0,C 180,E1 -11258.922,E2 -11258.922} C_VEL
LIN {X 0,Y 396.98,Z 449.662,A -85,B 0,C 180,E1 -11259.941,E2 -11259.941} C_VEL
LIN {X 0,Y 397.515,Z 442.414,A -85,B 0,C 180,E1 -11260.957,E2 -11260.957} C_VEL
LIN {X 0,Y 398.009,Z 434.711,A -85,B 0,C 180,E1 -11261.847,E2 -11261.847} C_VEL
LIN {X 0,Y 398.563,Z 426.664,A -85,B 0,C 180,E1 -11262.605,E2 -11262.605} C_VEL
LIN {X 0,Y 398.703,Z 420.229,A -85,B 0,C 180,E1 -11263.119,E2 -11263.119} C_VEL
LIN {X 0,Y 398.205,Z 411.649,A -85,B 0,C 180,E1 -11263.697,E2 -11263.697} C_VEL
LIN {X 0,Y 397.142,Z 401.996,A -85,B 0,C 180,E1 -11264.214,E2 -11264.214} C_VEL
LIN {X 0,Y 396.099,Z 394.458,A -85,B 0,C 180,E1 -11264.548,E2 -11264.548} C_VEL
LIN {X 0,Y 396.405,Z 386.315,A -85,B 0,C 180,E1 -11268.076,E2 -11268.076} C_VEL
LIN {X 0,Y 396.786,Z 377.873,A -85,B 0,C 180,E1 -11271.838,E2 -11271.838} C_VEL
LIN {X 0,Y 397.331,Z 369.773,A -85,B 0,C 180,E1 -11275.565,E2 -11275.565} C_VEL
LIN {X 0,Y 397.936,Z 362.483,A -85,B 0,C 180,E1 -11279.058,E2 -11279.058} C_VEL
LIN {X 0,Y 398.607,Z 356.235,A -85,B 0,C 180,E1 -11282.187,E2 -11282.187} C_VEL
LIN {X 0,Y 398.632,Z 352.754,A -85,B 0,C 180,E1 -11284.042,E2 -11284.042} C_VEL
LIN {X 0,Y 397.682,Z 347.085,A -85,B 0,C 180,E1 -11287.32,E2 -11287.32} C_VEL
LIN {X 0,Y 397.177,Z 343.83,A -85,B 0,C 180,E1 -11289.373,E2 -11289.373} C_VEL
LIN {X 0,Y 397.109,Z 343.84,A -85,B 0,C 180,E1 -11293.479,E2 -11293.479} C_VEL
LIN {X 0,Y 397.109,Z 343.837,A -85,B 0,C 180,E1 -11296.521,E2 -11296.521} C_VEL
LIN {X 0,Y 397.119,Z 343.832,A -85,B 0,C 180,E1 -11300.423,E2 -11300.423} C_VEL
LIN {X 0,Y 397.115,Z 343.833,A -85,B 0,C 180,E1 -11304.265,E2 -11304.265} C_VEL
LIN {X 0,Y 397.122,Z 343.832,A -85,B 0,C 180,E1 -11306.727,E2 -11306.727} C_VEL
LIN {X 0,Y 397.132,Z 343.831,A -85,B 0,C 180,E1 -11310.296,E2 -11310.296} C_VEL
LIN {X 0,Y 397.202,Z 343.822,A -85,B 0,C 180,E1 -11312.61,E2 -11312.61} C_VEL
LIN {X 0,Y 397.14,Z 343.829,A -85,B 0,C 180,E1 -11315.981,E2 -11315.981} C_VEL
LIN {X 0,Y 397.146,Z 343.829,A -85,B 0,C 180,E1 -11319.704,E2 -11319.704} C_VEL
LIN {X 0,Y 397.189,Z 343.822,A -85,B 0,C 180,E1 -11322.844,E2 -11322.844} C_VEL
LIN {X 0,Y 397.236,Z 343.817,A -85,B 0,C 180,E1 -11326.702,E2 -11326.702} C_VEL
LIN {X 0,Y 397.223,Z 343.819,A -85,B 0,C 180,E1 -11329.808,E2 -11329.808} C_VEL
LIN {X 0,Y 397.324,Z 343.808,A -85,B 0,C 180,E1 -11332.887,E2 -11332.887} C_VEL
LIN {X 0,Y 397.25,Z 343.816,A -85,B 0,C 180,E1 -11334.924,E2 -11334.924} C_VEL
LIN {X 0,Y 397.453,Z 343.789,A -85,B 0,C 180,E1 -11337.972,E2 -11337.972} C_VEL
LIN {X 0,Y 397.584,Z 343.776,A -85,B 0,C 180,E1 -11339.999,E2 -11339.999} C_VEL
LIN {X 0,Y 397.379,Z 343.799,A -85,B 0,C 180,E1 -11343.04,E2 -11343.04} C_VEL
LIN {X 0,Y 397.338,Z 343.804,A -85,B 0,C 180,E1 -11346.621,E2 -11346.621} C_VEL
LIN {X 0,Y 397.24,Z 343.817,A -85,B 0,C 180,E1 -11349.161,E2 -11349.161} C_VEL
LIN {X 0,Y 397.223,Z 343.82,A -85,B 0,C 180,E1 -11352.257,E2 -11352.257} C_VEL
LIN {X 0,Y 397.175,Z 343.831,A -85,B 0,C 180,E1 -11355.391,E2 -11355.391} C_VEL
LIN {X 0,Y 397.019,Z 343.849,A -85,B 0,C 180,E1 -11357.512,E2 -11357.512} C_VEL
LIN {X 0,Y 396.787,Z 344.26,A -85,B 0,C 180,E1 -11359.665,E2 -11359.665} C_VEL
LIN {X 0,Y 396.632,Z 347.727,A -85,B 0,C 180,E1 -11362.942,E2 -11362.942} C_VEL
LIN {X 0,Y 396.434,Z 351.373,A -85,B 0,C 180,E1 -11366.307,E2 -11366.307} C_VEL
LIN {X 0,Y 396.279,Z 355.213,A -85,B 0,C 180,E1 -11369.772,E2 -11369.772} C_VEL
LIN {X 0,Y 396.164,Z 359.474,A -85,B 0,C 180,E1 -11373.509,E2 -11373.509} C_VEL
LIN {X 0,Y 396.053,Z 361.857,A -85,B 0,C 180,E1 -11375.581,E2 -11375.581} C_VEL
LIN {X 0,Y 398.539,Z 373.427,A -85,B 0,C 180,E1 -11376.209,E2 -11376.209} C_VEL
LIN {X 0,Y 399.798,Z 380.783,A -85,B 0,C 180,E1 -11376.702,E2 -11376.702} C_VEL
LIN {X 0,Y 399.346,Z 389.697,A -85,B 0,C 180,E1 -11377.366,E2 -11377.366} C_VEL
LIN {X 0,Y 398.876,Z 397.332,A -85,B 0,C 180,E1 -11378.072,E2 -11378.072} C_VEL
LIN {X 0,Y 398.407,Z 403.665,A -85,B 0,C 180,E1 -11378.771,E2 -11378.771} C_VEL
LIN {X 0,Y 397.939,Z 410.823,A -85,B 0,C 180,E1 -11379.728,E2 -11379.728} C_VEL
LIN {X 0,Y 397.448,Z 417.745,A -85,B 0,C 180,E1 -11380.862,E2 -11380.862} C_VEL
LIN {X 0,Y 396.998,Z 423.259,A -85,B 0,C 180,E1 -11381.966,E2 -11381.966} C_VEL
LIN {X 0,Y 396.627,Z 427.528,A -85,B 0,C 180,E1 -11383.005,E2 -11383.005} C_VEL
LIN {X 0,Y 396.351,Z 431.697,A -85,B 0,C 180,E1 -11384.267,E2 -11384.267} C_VEL
LIN {X 0,Y 396.178,Z 434.154,A -85,B 0,C 180,E1 -11385.199,E2 -11385.199} C_VEL
LIN {X 0,Y 395.906,Z 437.065,A -85,B 0,C 180,E1 -11386.702,E2 -11386.702} C_VEL
LIN {X 0,Y 395.763,Z 438.86,A -85,B 0,C 180,E1 -11388.229,E2 -11388.229} C_VEL
LIN {X 0,Y 395.698,Z 439.549,A -85,B 0,C 180,E1 -11389.791,E2 -11389.791} C_VEL
LIN {X 0,Y 395.727,Z 438.805,A -85,B 0,C 180,E1 -11391.566,E2 -11391.566} C_VEL
LIN {X 0,Y 395.842,Z 437.052,A -85,B 0,C 180,E1 -11393.028,E2 -11393.028} C_VEL
LIN {X 0,Y 396.022,Z 434.988,A -85,B 0,C 180,E1 -11394.151,E2 -11394.151} C_VEL
LIN {X 0,Y 396.274,Z 430.165,A -85,B 0,C 180,E1 -11395.965,E2 -11395.965} C_VEL
LIN {X 0,Y 396.687,Z 424.024,A -85,B 0,C 180,E1 -11397.592,E2 -11397.592} C_VEL
LIN {X 0,Y 397.092,Z 417.971,A -85,B 0,C 180,E1 -11398.822,E2 -11398.822} C_VEL
LIN {X 0,Y 397.507,Z 411.739,A -85,B 0,C 180,E1 -11399.856,E2 -11399.856} C_VEL
LIN {X 0,Y 397.91,Z 404.918,A -85,B 0,C 180,E1 -11400.795,E2 -11400.795} C_VEL
LIN {X 0,Y 398.319,Z 398.361,A -85,B 0,C 180,E1 -11401.549,E2 -11401.549} C_VEL
LIN {X 0,Y 398.774,Z 390.301,A -85,B 0,C 180,E1 -11402.315,E2 -11402.315} C_VEL
LIN {X 0,Y 399.178,Z 381.73,A -85,B 0,C 180,E1 -11402.969,E2 -11402.969} C_VEL
LIN {X 0,Y 398.878,Z 376.856,A -85,B 0,C 180,E1 -11403.3,E2 -11403.3} C_VEL
LIN {X 0,Y 397.082,Z 366.573,A -85,B 0,C 180,E1 -11403.878,E2 -11403.878} C_VEL
LIN {X 0,Y 396.009,Z 360.965,A -85,B 0,C 180,E1 -11404.155,E2 -11404.155} C_VEL
LIN {X 0,Y 396.038,Z 357.103,A -85,B 0,C 180,E1 -11407.332,E2 -11407.332} C_VEL
LIN {X 0,Y 396.15,Z 353.56,A -85,B 0,C 180,E1 -11410.3,E2 -11410.3} C_VEL
LIN {X 0,Y 396.319,Z 349.759,A -85,B 0,C 180,E1 -11413.516,E2 -11413.516} C_VEL
LIN {X 0,Y 396.48,Z 345.564,A -85,B 0,C 180,E1 -11417.136,E2 -11417.136} C_VEL
LIN {X 0,Y 396.555,Z 343.904,A -85,B 0,C 180,E1 -11418.757,E2 -11418.757} C_VEL
LIN {X 0,Y 397.199,Z 343.824,A -85,B 0,C 180,E1 -11422.234,E2 -11422.234} C_VEL
LIN {X 0,Y 397.336,Z 343.805,A -85,B 0,C 180,E1 -11423.907,E2 -11423.907} C_VEL
LIN {X 0,Y 397.442,Z 343.792,A -85,B 0,C 180,E1 -11427.972,E2 -11427.972} C_VEL
LIN {X 0,Y 397.57,Z 343.777,A -85,B 0,C 180,E1 -11429.999,E2 -11429.999} C_VEL
LIN {X 0,Y 397.373,Z 343.798,A -85,B 0,C 180,E1 -11433.04,E2 -11433.04} C_VEL
LIN {X 0,Y 397.377,Z 343.801,A -85,B 0,C 180,E1 -11436.09,E2 -11436.09} C_VEL
LIN {X 0,Y 397.366,Z 343.802,A -85,B 0,C 180,E1 -11438.133,E2 -11438.133} C_VEL
LIN {X 0,Y 397.217,Z 343.819,A -85,B 0,C 180,E1 -11442.257,E2 -11442.257} C_VEL
LIN {X 0,Y 397.145,Z 343.826,A -85,B 0,C 180,E1 -11445.859,E2 -11445.859} C_VEL
LIN {X 0,Y 396.473,Z 343.911,A -85,B 0,C 180,E1 -11446.705,E2 -11446.705} C_VEL
LIN {X 0,Y 393.621,Z 344.267,A -85,B 0,C 180,E1 -11448.081,E2 -11448.081} C_VEL
LIN {X 0,Y 391.205,Z 344.569,A -85,B 0,C 180,E1 -11449.193,E2 -11449.193} C_VEL
LIN {X 0,Y 390.164,Z 344.698,A -85,B 0,C 180,E1 -11450.052,E2 -11450.052} C_VEL
LIN {X 0,Y 390.076,Z 344.707,A -85,B 0,C 180,E1 -11450.343,E2 -11450.343} C_VEL
LIN {X 0,Y 390.076,Z 344.71,A -85,B 0,C 180,E1 -11453.35,E2 -11453.35} C_VEL
LIN {X 0,Y 390.1,Z 344.704,A -85,B 0,C 180,E1 -11456.767,E2 -11456.767} C_VEL
LIN {X 0,Y 390.03,Z 344.712,A -85,B 0,C 180,E1 -11460.299,E2 -11460.299} C_VEL
LIN {X 0,Y 390.053,Z 344.709,A -85,B 0,C 180,E1 -11464.024,E2 -11464.024} C_VEL
LIN {X 0,Y 390.046,Z 344.713,A -85,B 0,C 180,E1 -11467.554,E2 -11467.554} C_VEL
LIN {X 0,Y 390.068,Z 344.71,A -85,B 0,C 180,E1 -11470.826,E2 -11470.826} C_VEL
LIN {X 0,Y 390.112,Z 344.702,A -85,B 0,C 180,E1 -11473.897,E2 -11473.897} C_VEL
LIN {X 0,Y 390.099,Z 344.707,A -85,B 0,C 180,E1 -11476.797,E2 -11476.797} C_VEL
LIN {X 0,Y 390.063,Z 344.708,A -85,B 0,C 180,E1 -11479.563,E2 -11479.563} C_VEL
LIN {X 0,Y 390.033,Z 344.715,A -85,B 0,C 180,E1 -11482.448,E2 -11482.448} C_VEL
LIN {X 0,Y 390.053,Z 344.71,A -85,B 0,C 180,E1 -11486.045,E2 -11486.045} C_VEL
LIN {X 0,Y 390.038,Z 344.711,A -85,B 0,C 180,E1 -11489.868,E2 -11489.868} C_VEL
LIN {X 0,Y 390.099,Z 344.704,A -85,B 0,C 180,E1 -11493.232,E2 -11493.232} C_VEL
LIN {X 0,Y 390.109,Z 344.706,A -85,B 0,C 180,E1 -11496.745,E2 -11496.745} C_VEL
LIN {X 0,Y 390.116,Z 344.703,A -85,B 0,C 180,E1 -11499.985,E2 -11499.985} C_VEL
LIN {X 0,Y 390.128,Z 344.7,A -85,B 0,C 180,E1 -11503.249,E2 -11503.249} C_VEL
LIN {X 0,Y 390.181,Z 344.696,A -85,B 0,C 180,E1 -11506.562,E2 -11506.562} C_VEL
LIN {X 0,Y 390.165,Z 344.696,A -85,B 0,C 180,E1 -11509.624,E2 -11509.624} C_VEL
LIN {X 0,Y 390.306,Z 344.679,A -85,B 0,C 180,E1 -11512.76,E2 -11512.76} C_VEL
LIN {X 0,Y 390.216,Z 344.689,A -85,B 0,C 180,E1 -11514.834,E2 -11514.834} C_VEL
LIN {X 0,Y 390.409,Z 344.669,A -85,B 0,C 180,E1 -11517.938,E2 -11517.938} C_VEL
LIN {X 0,Y 390.538,Z 344.653,A -85,B 0,C 180,E1 -11520.001,E2 -11520.001} C_VEL
LIN {X 0,Y 390.307,Z 344.678,A -85,B 0,C 180,E1 -11523.098,E2 -11523.098} C_VEL
LIN {X 0,Y 390.319,Z 344.679,A -85,B 0,C 180,E1 -11526.203,E2 -11526.203} C_VEL
LIN {X 0,Y 390.305,Z 344.679,A -85,B 0,C 180,E1 -11528.283,E2 -11528.283} C_VEL
LIN {X 0,Y 390.168,Z 344.695,A -85,B 0,C 180,E1 -11532.484,E2 -11532.484} C_VEL
LIN {X 0,Y 390.13,Z 344.703,A -85,B 0,C 180,E1 -11535.678,E2 -11535.678} C_VEL
LIN {X 0,Y 390.096,Z 344.705,A -85,B 0,C 180,E1 -11538.923,E2 -11538.923} C_VEL
LIN {X 0,Y 390.031,Z 344.713,A -85,B 0,C 180,E1 -11542.235,E2 -11542.235} C_VEL
LIN {X 0,Y 390.111,Z 344.705,A -85,B 0,C 180,E1 -11545.745,E2 -11545.745} C_VEL
LIN {X 0,Y 390.058,Z 344.712,A -85,B 0,C 180,E1 -11549.11,E2 -11549.11} C_VEL
LIN {X 0,Y 390.036,Z 344.714,A -85,B 0,C 180,E1 -11552.723,E2 -11552.723} C_VEL
LIN {X 0,Y 390.05,Z 344.71,A -85,B 0,C 180,E1 -11555.827,E2 -11555.827} C_VEL
LIN {X 0,Y 390.065,Z 344.712,A -85,B 0,C 180,E1 -11559.22,E2 -11559.22} C_VEL
LIN {X 0,Y 390.038,Z 344.713,A -85,B 0,C 180,E1 -11562.376,E2 -11562.376} C_VEL
LIN {X 0,Y 390.043,Z 344.712,A -85,B 0,C 180,E1 -11565.357,E2 -11565.357} C_VEL
LIN {X 0,Y 390.028,Z 344.714,A -85,B 0,C 180,E1 -11568.189,E2 -11568.189} C_VEL
LIN {X 0,Y 390.101,Z 344.859,A -85,B 0,C 180,E1 -11571.573,E2 -11571.573} C_VEL
LIN {X 0,Y 391.222,Z 350.95,A -85,B 0,C 180,E1 -11574.912,E2 -11574.912} C_VEL
LIN {X 0,Y 391.575,Z 354.586,A -85,B 0,C 180,E1 -11576.812,E2 -11576.812} C_VEL
LIN {X 0,Y 391.079,Z 360.631,A -85,B 0,C 180,E1 -11579.791,E2 -11579.791} C_VEL
LIN {X 0,Y 390.434,Z 367.879,A -85,B 0,C 180,E1 -11583.257,E2 -11583.257} C_VEL
LIN {X 0,Y 389.894,Z 375.541,A -85,B 0,C 180,E1 -11586.824,E2 -11586.824} C_VEL
LIN {X 0,Y 389.509,Z 382.427,A -85,B 0,C 180,E1 -11589.953,E2 -11589.953} C_VEL
LIN {X 0,Y 389.135,Z 390.874,A -85,B 0,C 180,E1 -11593.745,E2 -11593.745} C_VEL
LIN {X 0,Y 388.98,Z 395.039,A -85,B 0,C 180,E1 -11595.588,E2 -11595.588} C_VEL
LIN {X 0,Y 390.37,Z 407.137,A -85,B 0,C 180,E1 -11596.12,E2 -11596.12} C_VEL
LIN {X 0,Y 391.222,Z 417.713,A -85,B 0,C 180,E1 -11596.777,E2 -11596.777} C_VEL
LIN {X 0,Y 391.379,Z 424.629,A -85,B 0,C 180,E1 -11597.299,E2 -11597.299} C_VEL
LIN {X 0,Y 390.835,Z 433.035,A -85,B 0,C 180,E1 -11598.067,E2 -11598.067} C_VEL
LIN {X 0,Y 390.357,Z 441.046,A -85,B 0,C 180,E1 -11598.973,E2 -11598.973} C_VEL
LIN {X 0,Y 389.794,Z 449.383,A -85,B 0,C 180,E1 -11600.139,E2 -11600.139} C_VEL
LIN {X 0,Y 389.363,Z 456.811,A -85,B 0,C 180,E1 -11601.438,E2 -11601.438} C_VEL
LIN {X 0,Y 389.037,Z 462.617,A -85,B 0,C 180,E1 -11602.737,E2 -11602.737} C_VEL
LIN {X 0,Y 388.788,Z 467.566,A -85,B 0,C 180,E1 -11604.16,E2 -11604.16} C_VEL
LIN {X 0,Y 388.811,Z 470.762,A -85,B 0,C 180,E1 -11605.336,E2 -11605.336} C_VEL
LIN {X 0,Y 388.708,Z 473.788,A -85,B 0,C 180,E1 -11606.892,E2 -11606.892} C_VEL
LIN {X 0,Y 388.794,Z 475.152,A -85,B 0,C 180,E1 -11607.929,E2 -11607.929} C_VEL
LIN {X 0,Y 388.76,Z 476.02,A -85,B 0,C 180,E1 -11608.965,E2 -11608.965} C_VEL
LIN {X 0,Y 388.746,Z 476.319,A -85,B 0,C 180,E1 -11610.001,E2 -11610.001} C_VEL
LIN {X 0,Y 388.76,Z 476.07,A -85,B 0,C 180,E1 -11611.037,E2 -11611.037} C_VEL
LIN {X 0,Y 388.76,Z 475.35,A -85,B 0,C 180,E1 -11612.073,E2 -11612.073} C_VEL
LIN {X 0,Y 388.692,Z 474.147,A -85,B 0,C 180,E1 -11613.111,E2 -11613.111} C_VEL
LIN {X 0,Y 388.811,Z 471.266,A -85,B 0,C 180,E1 -11614.667,E2 -11614.667} C_VEL
LIN {X 0,Y 388.836,Z 467.11,A -85,B 0,C 180,E1 -11616.227,E2 -11616.227} C_VEL
LIN {X 0,Y 389.196,Z 461.53,A -85,B 0,C 180,E1 -11617.785,E2 -11617.785} C_VEL
LIN {X 0,Y 389.535,Z 455.428,A -85,B 0,C 180,E1 -11619.084,E2 -11619.084} C_VEL
LIN {X 0,Y 389.978,Z 449.492,A -85,B 0,C 180,E1 -11620.121,E2 -11620.121} C_VEL
LIN {X 0,Y 390.539,Z 442.29,A -85,B 0,C 180,E1 -11621.156,E2 -11621.156} C_VEL
LIN {X 0,Y 391.061,Z 434.638,A -85,B 0,C 180,E1 -11622.06,E2 -11622.06} C_VEL
LIN {X 0,Y 391.638,Z 426.65,A -85,B 0,C 180,E1 -11622.832,E2 -11622.832} C_VEL
LIN {X 0,Y 391.723,Z 420.298,A -85,B 0,C 180,E1 -11623.357,E2 -11623.357} C_VEL
LIN {X 0,Y 391.16,Z 410.638,A -85,B 0,C 180,E1 -11624.016,E2 -11624.016} C_VEL
LIN {X 0,Y 390.028,Z 401.177,A -85,B 0,C 180,E1 -11624.53,E2 -11624.53} C_VEL
LIN {X 0,Y 389.034,Z 394.124,A -85,B 0,C 180,E1 -11624.852,E2 -11624.852} C_VEL
LIN {X 0,Y 389.333,Z 386.09,A -85,B 0,C 180,E1 -11628.416,E2 -11628.416} C_VEL
LIN {X 0,Y 389.703,Z 378.875,A -85,B 0,C 180,E1 -11631.698,E2 -11631.698} C_VEL
LIN {X 0,Y 390.186,Z 371.734,A -85,B 0,C 180,E1 -11635.043,E2 -11635.043} C_VEL
LIN {X 0,Y 390.75,Z 365.243,A -85,B 0,C 180,E1 -11638.198,E2 -11638.198} C_VEL
LIN {X 0,Y 391.552,Z 357.871,A -85,B 0,C 180,E1 -11641.934,E2 -11641.934} C_VEL
LIN {X 0,Y 391.677,Z 354.402,A -85,B 0,C 180,E1 -11643.798,E2 -11643.798} C_VEL
LIN {X 0,Y 390.803,Z 348.915,A -85,B 0,C 180,E1 -11647.017,E2 -11647.017} C_VEL
LIN {X 0,Y 390.108,Z 344.712,A -85,B 0,C 180,E1 -11649.79,E2 -11649.79} C_VEL
LIN {X 0,Y 390.064,Z 344.718,A -85,B 0,C 180,E1 -11653.211,E2 -11653.211} C_VEL
LIN {X 0,Y 390.064,Z 344.712,A -85,B 0,C 180,E1 -11656.79,E2 -11656.79} C_VEL
LIN {X 0,Y 390.064,Z 344.712,A -85,B 0,C 180,E1 -11659.561,E2 -11659.561} C_VEL
LIN {X 0,Y 390.049,Z 344.714,A -85,B 0,C 180,E1 -11662.45,E2 -11662.45} C_VEL
LIN {X 0,Y 390.076,Z 344.71,A -85,B 0,C 180,E1 -11665.975,E2 -11665.975} C_VEL
LIN {X 0,Y 390.054,Z 344.712,A -85,B 0,C 180,E1 -11669.869,E2 -11669.869} C_VEL
LIN {X 0,Y 390.121,Z 344.704,A -85,B 0,C 180,E1 -11673.232,E2 -11673.232} C_VEL
LIN {X 0,Y 390.114,Z 344.704,A -85,B 0,C 180,E1 -11676.75,E2 -11676.75} C_VEL
LIN {X 0,Y 390.111,Z 344.705,A -85,B 0,C 180,E1 -11679.983,E2 -11679.983} C_VEL
LIN {X 0,Y 390.145,Z 344.7,A -85,B 0,C 180,E1 -11683.248,E2 -11683.248} C_VEL
LIN {X 0,Y 390.202,Z 344.693,A -85,B 0,C 180,E1 -11686.561,E2 -11686.561} C_VEL
LIN {X 0,Y 390.174,Z 344.698,A -85,B 0,C 180,E1 -11689.622,E2 -11689.622} C_VEL
LIN {X 0,Y 390.273,Z 344.685,A -85,B 0,C 180,E1 -11692.757,E2 -11692.757} C_VEL
LIN {X 0,Y 390.221,Z 344.691,A -85,B 0,C 180,E1 -11694.832,E2 -11694.832} C_VEL
LIN {X 0,Y 390.422,Z 344.665,A -85,B 0,C 180,E1 -11697.936,E2 -11697.936} C_VEL
LIN {X 0,Y 390.554,Z 344.651,A -85,B 0,C 180,E1 -11699.999,E2 -11699.999} C_VEL
LIN {X 0,Y 390.313,Z 344.679,A -85,B 0,C 180,E1 -11703.095,E2 -11703.095} C_VEL
LIN {X 0,Y 390.293,Z 344.681,A -85,B 0,C 180,E1 -11706.614,E2 -11706.614} C_VEL
LIN {X 0,Y 390.197,Z 344.694,A -85,B 0,C 180,E1 -11709.328,E2 -11709.328} C_VEL
LIN {X 0,Y 390.175,Z 344.698,A -85,B 0,C 180,E1 -11712.482,E2 -11712.482} C_VEL
LIN {X 0,Y 390.128,Z 344.708,A -85,B 0,C 180,E1 -11715.676,E2 -11715.676} C_VEL
LIN {X 0,Y 389.916,Z 344.733,A -85,B 0,C 180,E1 -11717.842,E2 -11717.842} C_VEL
LIN {X 0,Y 389.799,Z 344.746,A -85,B 0,C 180,E1 -11718.936,E2 -11718.936} C_VEL
LIN {X 0,Y 389.673,Z 346.734,A -85,B 0,C 180,E1 -11721.143,E2 -11721.143} C_VEL
LIN {X 0,Y 389.489,Z 350.311,A -85,B 0,C 180,E1 -11724.519,E2 -11724.519} C_VEL
LIN {X 0,Y 389.285,Z 354.071,A -85,B 0,C 180,E1 -11727.993,E2 -11727.993} C_VEL
LIN {X 0,Y 389.168,Z 358.031,A -85,B 0,C 180,E1 -11731.58,E2 -11731.58} C_VEL
LIN {X 0,Y 389,Z 362.228,A -85,B 0,C 180,E1 -11735.278,E2 -11735.278} C_VEL
LIN {X 0,Y 391.498,Z 373.517,A -85,B 0,C 180,E1 -11735.909,E2 -11735.909} C_VEL
LIN {X 0,Y 392.905,Z 381.935,A -85,B 0,C 180,E1 -11736.493,E2 -11736.493} C_VEL
LIN {X 0,Y 392.44,Z 390.871,A -85,B 0,C 180,E1 -11737.184,E2 -11737.184} C_VEL
LIN {X 0,Y 391.939,Z 398.413,A -85,B 0,C 180,E1 -11737.908,E2 -11737.908} C_VEL
LIN {X 0,Y 391.444,Z 404.982,A -85,B 0,C 180,E1 -11738.666,E2 -11738.666} C_VEL
LIN {X 0,Y 390.959,Z 411.583,A -85,B 0,C 180,E1 -11739.578,E2 -11739.578} C_VEL
LIN {X 0,Y 390.49,Z 417.848,A -85,B 0,C 180,E1 -11740.623,E2 -11740.623} C_VEL
LIN {X 0,Y 389.998,Z 423.709,A -85,B 0,C 180,E1 -11741.816,E2 -11741.816} C_VEL
LIN {X 0,Y 389.612,Z 427.848,A -85,B 0,C 180,E1 -11742.842,E2 -11742.842} C_VEL
LIN {X 0,Y 389.285,Z 432.566,A -85,B 0,C 180,E1 -11744.318,E2 -11744.318} C_VEL
LIN {X 0,Y 389.018,Z 436.046,A -85,B 0,C 180,E1 -11745.795,E2 -11745.795} C_VEL
LIN {X 0,Y 388.837,Z 437.41,A -85,B 0,C 180,E1 -11746.619,E2 -11746.619} C_VEL
LIN {X 0,Y 388.689,Z 439.052,A -85,B 0,C 180,E1 -11748.008,E2 -11748.008} C_VEL
LIN {X 0,Y 388.614,Z 439.791,A -85,B 0,C 180,E1 -11749.423,E2 -11749.423} C_VEL
LIN {X 0,Y 388.605,Z 439.533,A -85,B 0,C 180,E1 -11751.045,E2 -11751.045} C_VEL
LIN {X 0,Y 388.734,Z 437.955,A -85,B 0,C 180,E1 -11752.698,E2 -11752.698} C_VEL
LIN {X 0,Y 388.949,Z 434.876,A -85,B 0,C 180,E1 -11754.399,E2 -11754.399} C_VEL
LIN {X 0,Y 389.186,Z 430.765,A -85,B 0,C 180,E1 -11755.957,E2 -11755.957} C_VEL
LIN {X 0,Y 389.62,Z 424.718,A -85,B 0,C 180,E1 -11757.623,E2 -11757.623} C_VEL
LIN {X 0,Y 390.003,Z 419.18,A -85,B 0,C 180,E1 -11758.795,E2 -11758.795} C_VEL
LIN {X 0,Y 390.538,Z 411.701,A -85,B 0,C 180,E1 -11760.063,E2 -11760.063} C_VEL
LIN {X 0,Y 390.915,Z 405.278,A -85,B 0,C 180,E1 -11760.959,E2 -11760.959} C_VEL
LIN {X 0,Y 391.436,Z 396.926,A -85,B 0,C 180,E1 -11761.917,E2 -11761.917} C_VEL
LIN {X 0,Y 391.968,Z 387.382,A -85,B 0,C 180,E1 -11762.791,E2 -11762.791} C_VEL
LIN {X 0,Y 392.152,Z 379.208,A -85,B 0,C 180,E1 -11763.381,E2 -11763.381} C_VEL
LIN {X 0,Y 390.185,Z 367.758,A -85,B 0,C 180,E1 -11764.064,E2 -11764.064} C_VEL
LIN {X 0,Y 388.944,Z 361.252,A -85,B 0,C 180,E1 -11764.401,E2 -11764.401} C_VEL
LIN {X 0,Y 388.982,Z 357.294,A -85,B 0,C 180,E1 -11767.701,E2 -11767.701} C_VEL
LIN {X 0,Y 389.088,Z 353.363,A -85,B 0,C 180,E1 -11771.025,E2 -11771.025} C_VEL
LIN {X 0,Y 389.249,Z 349.588,A -85,B 0,C 180,E1 -11774.285,E2 -11774.285} C_VEL
LIN {X 0,Y 389.436,Z 345.918,A -85,B 0,C 180,E1 -11777.492,E2 -11777.492} C_VEL
LIN {X 0,Y 389.49,Z 344.785,A -85,B 0,C 180,E1 -11778.55,E2 -11778.55} C_VEL
LIN {X 0,Y 390.154,Z 344.701,A -85,B 0,C 180,E1 -11782.183,E2 -11782.183} C_VEL
LIN {X 0,Y 390.211,Z 344.69,A -85,B 0,C 180,E1 -11784.832,E2 -11784.832} C_VEL
LIN {X 0,Y 390.411,Z 344.668,A -85,B 0,C 180,E1 -11787.935,E2 -11787.935} C_VEL
LIN {X 0,Y 390.539,Z 344.653,A -85,B 0,C 180,E1 -11789.999,E2 -11789.999} C_VEL
LIN {X 0,Y 390.307,Z 344.678,A -85,B 0,C 180,E1 -11793.095,E2 -11793.095} C_VEL
LIN {X 0,Y 390.33,Z 344.678,A -85,B 0,C 180,E1 -11796.2,E2 -11796.2} C_VEL
LIN {X 0,Y 390.303,Z 344.68,A -85,B 0,C 180,E1 -11798.281,E2 -11798.281} C_VEL
LIN {X 0,Y 390.166,Z 344.696,A -85,B 0,C 180,E1 -11802.482,E2 -11802.482} C_VEL
LIN {X 0,Y 390.117,Z 344.704,A -85,B 0,C 180,E1 -11805.852,E2 -11805.852} C_VEL
LIN {X 0,Y 390.092,Z 344.705,A -85,B 0,C 180,E1 -11808.921,E2 -11808.921} C_VEL
LIN {X 0,Y 390.076,Z 344.707,A -85,B 0,C 180,E1 -11810.343,E2 -11810.343} C_VEL
LIN {X 0,Y 389.39,Z 344.795,A -85,B 0,C 180,E1 -11811.205,E2 -11811.205} C_VEL
LIN {X 0,Y 386.503,Z 345.152,A -85,B 0,C 180,E1 -11812.606,E2 -11812.606} C_VEL
LIN {X 0,Y 384.092,Z 345.456,A -85,B 0,C 180,E1 -11813.738,E2 -11813.738} C_VEL
LIN {X 0,Y 383.095,Z 345.576,A -85,B 0,C 180,E1 -11814.614,E2 -11814.614} C_VEL
LIN {X 0,Y 383.034,Z 345.584,A -85,B 0,C 180,E1 -11814.911,E2 -11814.911} C_VEL
LIN {X 0,Y 383.035,Z 345.583,A -85,B 0,C 180,E1 -11818.491,E2 -11818.491} C_VEL
LIN {X 0,Y 382.997,Z 345.589,A -85,B 0,C 180,E1 -11822.149,E2 -11822.149} C_VEL
LIN {X 0,Y 383.004,Z 345.588,A -85,B 0,C 180,E1 -11824.667,E2 -11824.667} C_VEL
LIN {X 0,Y 382.995,Z 345.589,A -85,B 0,C 180,E1 -11827.905,E2 -11827.905} C_VEL
LIN {X 0,Y 383.032,Z 345.587,A -85,B 0,C 180,E1 -11831.339,E2 -11831.339} C_VEL
LIN {X 0,Y 383.054,Z 345.581,A -85,B 0,C 180,E1 -11834.314,E2 -11834.314} C_VEL
LIN {X 0,Y 383.06,Z 345.583,A -85,B 0,C 180,E1 -11837.249,E2 -11837.249} C_VEL
LIN {X 0,Y 383.008,Z 345.588,A -85,B 0,C 180,E1 -11840.412,E2 -11840.412} C_VEL
LIN {X 0,Y 383.012,Z 345.586,A -85,B 0,C 180,E1 -11844.045,E2 -11844.045} C_VEL
LIN {X 0,Y 382.975,Z 345.591,A -85,B 0,C 180,E1 -11847.577,E2 -11847.577} C_VEL
LIN {X 0,Y 382.984,Z 345.592,A -85,B 0,C 180,E1 -11850.301,E2 -11850.301} C_VEL
LIN {X 0,Y 383.042,Z 345.587,A -85,B 0,C 180,E1 -11852.699,E2 -11852.699} C_VEL
LIN {X 0,Y 383.034,Z 345.586,A -85,B 0,C 180,E1 -11856.194,E2 -11856.194} C_VEL
LIN {X 0,Y 383.068,Z 345.579,A -85,B 0,C 180,E1 -11859.601,E2 -11859.601} C_VEL
LIN {X 0,Y 383.094,Z 345.577,A -85,B 0,C 180,E1 -11862.932,E2 -11862.932} C_VEL
LIN {X 0,Y 383.113,Z 345.577,A -85,B 0,C 180,E1 -11866.464,E2 -11866.464} C_VEL
LIN {X 0,Y 383.128,Z 345.572,A -85,B 0,C 180,E1 -11869.431,E2 -11869.431} C_VEL
LIN {X 0,Y 383.261,Z 345.557,A -85,B 0,C 180,E1 -11872.626,E2 -11872.626} C_VEL
LIN {X 0,Y 383.188,Z 345.565,A -85,B 0,C 180,E1 -11874.739,E2 -11874.739} C_VEL
LIN {X 0,Y 383.376,Z 345.545,A -85,B 0,C 180,E1 -11877.9,E2 -11877.9} C_VEL
LIN {X 0,Y 383.508,Z 345.528,A -85,B 0,C 180,E1 -11880.001,E2 -11880.001} C_VEL
LIN {X 0,Y 383.244,Z 345.558,A -85,B 0,C 180,E1 -11883.155,E2 -11883.155} C_VEL
LIN {X 0,Y 383.277,Z 345.555,A -85,B 0,C 180,E1 -11886.317,E2 -11886.317} C_VEL
LIN {X 0,Y 383.25,Z 345.557,A -85,B 0,C 180,E1 -11888.437,E2 -11888.437} C_VEL
LIN {X 0,Y 383.098,Z 345.58,A -85,B 0,C 180,E1 -11891.643,E2 -11891.643} C_VEL
LIN {X 0,Y 383.102,Z 345.575,A -85,B 0,C 180,E1 -11894.883,E2 -11894.883} C_VEL
LIN {X 0,Y 383.054,Z 345.582,A -85,B 0,C 180,E1 -11898.175,E2 -11898.175} C_VEL
LIN {X 0,Y 382.984,Z 345.594,A -85,B 0,C 180,E1 -11901.532,E2 -11901.532} C_VEL
LIN {X 0,Y 383.044,Z 345.584,A -85,B 0,C 180,E1 -11904.962,E2 -11904.962} C_VEL
LIN {X 0,Y 383.042,Z 345.583,A -85,B 0,C 180,E1 -11908.493,E2 -11908.493} C_VEL
LIN {X 0,Y 383.004,Z 345.587,A -85,B 0,C 180,E1 -11912.151,E2 -11912.151} C_VEL
LIN {X 0,Y 383.011,Z 345.588,A -85,B 0,C 180,E1 -11914.669,E2 -11914.669} C_VEL
LIN {X 0,Y 382.995,Z 345.589,A -85,B 0,C 180,E1 -11917.906,E2 -11917.906} C_VEL
LIN {X 0,Y 382.979,Z 345.593,A -85,B 0,C 180,E1 -11921.349,E2 -11921.349} C_VEL
LIN {X 0,Y 382.994,Z 345.589,A -85,B 0,C 180,E1 -11924.305,E2 -11924.305} C_VEL
LIN {X 0,Y 383.005,Z 345.589,A -85,B 0,C 180,E1 -11927.242,E2 -11927.242} C_VEL
LIN {X 0,Y 383.07,Z 345.667,A -85,B 0,C 180,E1 -11931.325,E2 -11931.325} C_VEL
LIN {X 0,Y 384.169,Z 351.899,A -85,B 0,C 180,E1 -11934.815,E2 -11934.815} C_VEL
LIN {X 0,Y 384.551,Z 355.531,A -85,B 0,C 180,E1 -11936.753,E2 -11936.753} C_VEL
LIN {X 0,Y 384.116,Z 360.616,A -85,B 0,C 180,E1 -11939.311,E2 -11939.311} C_VEL
LIN {X 0,Y 383.469,Z 367.598,A -85,B 0,C 180,E1 -11942.732,E2 -11942.732} C_VEL
LIN {X 0,Y 382.911,Z 374.842,A -85,B 0,C 180,E1 -11946.186,E2 -11946.186} C_VEL
LIN {X 0,Y 382.459,Z 382.108,A -85,B 0,C 180,E1 -11949.582,E2 -11949.582} C_VEL
LIN {X 0,Y 382.11,Z 389.61,A -85,B 0,C 180,E1 -11953.023,E2 -11953.023} C_VEL
LIN {X 0,Y 381.923,Z 394.724,A -85,B 0,C 180,E1 -11955.335,E2 -11955.335} C_VEL
LIN {X 0,Y 383.424,Z 408.173,A -85,B 0,C 180,E1 -11955.973,E2 -11955.973} C_VEL
LIN {X 0,Y 384.191,Z 417.739,A -85,B 0,C 180,E1 -11956.588,E2 -11956.588} C_VEL
LIN {X 0,Y 384.349,Z 425.535,A -85,B 0,C 180,E1 -11957.204,E2 -11957.204} C_VEL
LIN {X 0,Y 383.777,Z 433.659,A -85,B 0,C 180,E1 -11957.978,E2 -11957.978} C_VEL
LIN {X 0,Y 383.296,Z 441.513,A -85,B 0,C 180,E1 -11958.901,E2 -11958.901} C_VEL
LIN {X 0,Y 382.786,Z 448.868,A -85,B 0,C 180,E1 -11959.957,E2 -11959.957} C_VEL
LIN {X 0,Y 382.307,Z 456.337,A -85,B 0,C 180,E1 -11961.278,E2 -11961.278} C_VEL
LIN {X 0,Y 381.967,Z 462.186,A -85,B 0,C 180,E1 -11962.601,E2 -11962.601} C_VEL
LIN {X 0,Y 381.739,Z 466.465,A -85,B 0,C 180,E1 -11963.812,E2 -11963.812} C_VEL
LIN {X 0,Y 381.717,Z 470.372,A -85,B 0,C 180,E1 -11965.249,E2 -11965.249} C_VEL
LIN {X 0,Y 381.615,Z 473.414,A -85,B 0,C 180,E1 -11966.834,E2 -11966.834} C_VEL
LIN {X 0,Y 381.693,Z 474.794,A -85,B 0,C 180,E1 -11967.891,E2 -11967.891} C_VEL
LIN {X 0,Y 381.692,Z 475.677,A -85,B 0,C 180,E1 -11968.946,E2 -11968.946} C_VEL
LIN {X 0,Y 381.676,Z 475.977,A -85,B 0,C 180,E1 -11970.001,E2 -11970.001} C_VEL
LIN {X 0,Y 381.691,Z 475.743,A -85,B 0,C 180,E1 -11971.056,E2 -11971.056} C_VEL
LIN {X 0,Y 381.659,Z 475.037,A -85,B 0,C 180,E1 -11972.112,E2 -11972.112} C_VEL
LIN {X 0,Y 381.601,Z 473.851,A -85,B 0,C 180,E1 -11973.169,E2 -11973.169} C_VEL
LIN {X 0,Y 381.717,Z 470.99,A -85,B 0,C 180,E1 -11974.754,E2 -11974.754} C_VEL
LIN {X 0,Y 381.772,Z 466.857,A -85,B 0,C 180,E1 -11976.343,E2 -11976.343} C_VEL
LIN {X 0,Y 382.135,Z 461.306,A -85,B 0,C 180,E1 -11977.93,E2 -11977.93} C_VEL
LIN {X 0,Y 382.514,Z 455.243,A -85,B 0,C 180,E1 -11979.253,E2 -11979.253} C_VEL
LIN {X 0,Y 382.982,Z 449.337,A -85,B 0,C 180,E1 -11980.308,E2 -11980.308} C_VEL
LIN {X 0,Y 383.548,Z 442.17,A -85,B 0,C 180,E1 -11981.362,E2 -11981.362} C_VEL
LIN {X 0,Y 384.125,Z 434.564,A -85,B 0,C 180,E1 -11982.281,E2 -11982.281} C_VEL
LIN {X 0,Y 384.718,Z 426.636,A -85,B 0,C 180,E1 -11983.067,E2 -11983.067} C_VEL
LIN {X 0,Y 384.703,Z 418.522,A -85,B 0,C 180,E1 -11983.74,E2 -11983.74} C_VEL
LIN {X 0,Y 384.028,Z 409.166,A -85,B 0,C 180,E1 -11984.378,E2 -11984.378} C_VEL
LIN {X 0,Y 382.714,Z 398.861,A -85,B 0,C 180,E1 -11984.933,E2 -11984.933} C_VEL
LIN {X 0,Y 381.995,Z 393.77,A -85,B 0,C 180,E1 -11985.166,E2 -11985.166} C_VEL
LIN {X 0,Y 382.281,Z 385.858,A -85,B 0,C 180,E1 -11988.769,E2 -11988.769} C_VEL
LIN {X 0,Y 382.689,Z 378.676,A -85,B 0,C 180,E1 -11992.117,E2 -11992.117} C_VEL
LIN {X 0,Y 383.222,Z 371.623,A -85,B 0,C 180,E1 -11995.502,E2 -11995.502} C_VEL
LIN {X 0,Y 383.841,Z 364.555,A -85,B 0,C 180,E1 -11999.027,E2 -11999.027} C_VEL
LIN {X 0,Y 384.554,Z 358.854,A -85,B 0,C 180,E1 -12002.006,E2 -12002.006} C_VEL
LIN {X 0,Y 384.667,Z 355.493,A -85,B 0,C 180,E1 -12003.867,E2 -12003.867} C_VEL
LIN {X 0,Y 383.793,Z 349.975,A -85,B 0,C 180,E1 -12007.179,E2 -12007.179} C_VEL
LIN {X 0,Y 383.035,Z 345.593,A -85,B 0,C 180,E1 -12010.128,E2 -12010.128} C_VEL
LIN {X 0,Y 383.013,Z 345.597,A -85,B 0,C 180,E1 -12012.779,E2 -12012.779} C_VEL
LIN {X 0,Y 383.004,Z 345.594,A -85,B 0,C 180,E1 -12015.789,E2 -12015.789} C_VEL
LIN {X 0,Y 382.995,Z 345.592,A -85,B 0,C 180,E1 -12018.796,E2 -12018.796} C_VEL
LIN {X 0,Y 383.005,Z 345.591,A -85,B 0,C 180,E1 -12022.097,E2 -12022.097} C_VEL
LIN {X 0,Y 383.025,Z 345.588,A -85,B 0,C 180,E1 -12025.332,E2 -12025.332} C_VEL
LIN {X 0,Y 382.99,Z 345.592,A -85,B 0,C 180,E1 -12029.081,E2 -12029.081} C_VEL
LIN {X 0,Y 383.064,Z 345.583,A -85,B 0,C 180,E1 -12032.698,E2 -12032.698} C_VEL
LIN {X 0,Y 383.041,Z 345.586,A -85,B 0,C 180,E1 -12036.192,E2 -12036.192} C_VEL
LIN {X 0,Y 383.063,Z 345.583,A -85,B 0,C 180,E1 -12039.598,E2 -12039.598} C_VEL
LIN {X 0,Y 383.113,Z 345.575,A -85,B 0,C 180,E1 -12042.931,E2 -12042.931} C_VEL
LIN {X 0,Y 383.133,Z 345.574,A -85,B 0,C 180,E1 -12046.463,E2 -12046.463} C_VEL
LIN {X 0,Y 383.15,Z 345.573,A -85,B 0,C 180,E1 -12050.497,E2 -12050.497} C_VEL
LIN {X 0,Y 383.261,Z 345.557,A -85,B 0,C 180,E1 -12053.682,E2 -12053.682} C_VEL
LIN {X 0,Y 383.389,Z 345.541,A -85,B 0,C 180,E1 -12057.898,E2 -12057.898} C_VEL
LIN {X 0,Y 383.523,Z 345.527,A -85,B 0,C 180,E1 -12059.999,E2 -12059.999} C_VEL
LIN {X 0,Y 383.25,Z 345.559,A -85,B 0,C 180,E1 -12063.153,E2 -12063.153} C_VEL
LIN {X 0,Y 383.253,Z 345.558,A -85,B 0,C 180,E1 -12066.604,E2 -12066.604} C_VEL
LIN {X 0,Y 383.148,Z 345.573,A -85,B 0,C 180,E1 -12069.501,E2 -12069.501} C_VEL
LIN {X 0,Y 383.13,Z 345.577,A -85,B 0,C 180,E1 -12073.535,E2 -12073.535} C_VEL
LIN {X 0,Y 383.014,Z 345.593,A -85,B 0,C 180,E1 -12077.072,E2 -12077.072} C_VEL
LIN {X 0,Y 382.714,Z 345.843,A -85,B 0,C 180,E1 -12079.301,E2 -12079.301} C_VEL
LIN {X 0,Y 382.55,Z 349.264,A -85,B 0,C 180,E1 -12082.692,E2 -12082.692} C_VEL
LIN {X 0,Y 382.339,Z 352.958,A -85,B 0,C 180,E1 -12086.176,E2 -12086.176} C_VEL
LIN {X 0,Y 382.169,Z 356.813,A -85,B 0,C 180,E1 -12089.769,E2 -12089.769} C_VEL
LIN {X 0,Y 382.002,Z 360.928,A -85,B 0,C 180,E1 -12093.498,E2 -12093.498} C_VEL
LIN {X 0,Y 381.956,Z 362.56,A -85,B 0,C 180,E1 -12094.957,E2 -12094.957} C_VEL
LIN {X 0,Y 384.557,Z 374.094,A -85,B 0,C 180,E1 -12095.627,E2 -12095.627} C_VEL
LIN {X 0,Y 386.036,Z 382.985,A -85,B 0,C 180,E1 -12096.269,E2 -12096.269} C_VEL
LIN {X 0,Y 385.598,Z 390.828,A -85,B 0,C 180,E1 -12096.887,E2 -12096.887} C_VEL
LIN {X 0,Y 385.022,Z 399.102,A -85,B 0,C 180,E1 -12097.696,E2 -12097.696} C_VEL
LIN {X 0,Y 384.541,Z 405.229,A -85,B 0,C 180,E1 -12098.416,E2 -12098.416} C_VEL
LIN {X 0,Y 383.99,Z 412.391,A -85,B 0,C 180,E1 -12099.43,E2 -12099.43} C_VEL
LIN {X 0,Y 383.462,Z 418.833,A -85,B 0,C 180,E1 -12100.541,E2 -12100.541} C_VEL
LIN {X 0,Y 382.847,Z 425.748,A -85,B 0,C 180,E1 -12102.021,E2 -12102.021} C_VEL
LIN {X 0,Y 382.425,Z 430.997,A -85,B 0,C 180,E1 -12103.509,E2 -12103.509} C_VEL
LIN {X 0,Y 382.063,Z 434.875,A -85,B 0,C 180,E1 -12104.98,E2 -12104.98} C_VEL
LIN {X 0,Y 381.914,Z 436.73,A -85,B 0,C 180,E1 -12105.861,E2 -12105.861} C_VEL
LIN {X 0,Y 381.645,Z 438.951,A -85,B 0,C 180,E1 -12107.44,E2 -12107.44} C_VEL
LIN {X 0,Y 381.53,Z 440.036,A -85,B 0,C 180,E1 -12109.044,E2 -12109.044} C_VEL
LIN {X 0,Y 381.503,Z 440.234,A -85,B 0,C 180,E1 -12109.851,E2 -12109.851} C_VEL
LIN {X 0,Y 381.519,Z 439.777,A -85,B 0,C 180,E1 -12111.22,E2 -12111.22} C_VEL
LIN {X 0,Y 381.644,Z 438.488,A -85,B 0,C 180,E1 -12112.575,E2 -12112.575} C_VEL
LIN {X 0,Y 381.826,Z 436.015,A -85,B 0,C 180,E1 -12114.081,E2 -12114.081} C_VEL
LIN {X 0,Y 381.986,Z 433.434,A -85,B 0,C 180,E1 -12115.224,E2 -12115.224} C_VEL
LIN {X 0,Y 382.341,Z 428.437,A -85,B 0,C 180,E1 -12116.835,E2 -12116.835} C_VEL
LIN {X 0,Y 382.706,Z 423.255,A -85,B 0,C 180,E1 -12118.131,E2 -12118.131} C_VEL
LIN {X 0,Y 383.143,Z 417.196,A -85,B 0,C 180,E1 -12119.351,E2 -12119.351} C_VEL
LIN {X 0,Y 383.719,Z 409.225,A -85,B 0,C 180,E1 -12120.645,E2 -12120.645} C_VEL
LIN {X 0,Y 384.281,Z 400.467,A -85,B 0,C 180,E1 -12121.755,E2 -12121.755} C_VEL
LIN {X 0,Y 384.742,Z 392.915,A -85,B 0,C 180,E1 -12122.532,E2 -12122.532} C_VEL
LIN {X 0,Y 385.218,Z 383.94,A -85,B 0,C 180,E1 -12123.272,E2 -12123.272} C_VEL
LIN {X 0,Y 385.061,Z 379.347,A -85,B 0,C 180,E1 -12123.609,E2 -12123.609} C_VEL
LIN {X 0,Y 383.073,Z 368.027,A -85,B 0,C 180,E1 -12124.297,E2 -12124.297} C_VEL
LIN {X 0,Y 381.89,Z 361.562,A -85,B 0,C 180,E1 -12124.634,E2 -12124.634} C_VEL
LIN {X 0,Y 381.92,Z 357.099,A -85,B 0,C 180,E1 -12128.404,E2 -12128.404} C_VEL
LIN {X 0,Y 382.06,Z 353.173,A -85,B 0,C 180,E1 -12131.776,E2 -12131.776} C_VEL
LIN {X 0,Y 382.202,Z 349.399,A -85,B 0,C 180,E1 -12135.081,E2 -12135.081} C_VEL
LIN {X 0,Y 382.431,Z 345.736,A -85,B 0,C 180,E1 -12138.336,E2 -12138.336} C_VEL
LIN {X 0,Y 383.094,Z 345.58,A -85,B 0,C 180,E1 -12142.146,E2 -12142.146} C_VEL
LIN {X 0,Y 383.181,Z 345.567,A -85,B 0,C 180,E1 -12144.737,E2 -12144.737} C_VEL
LIN {X 0,Y 383.378,Z 345.544,A -85,B 0,C 180,E1 -12147.898,E2 -12147.898} C_VEL
LIN {X 0,Y 383.509,Z 345.529,A -85,B 0,C 180,E1 -12149.999,E2 -12149.999} C_VEL
LIN {X 0,Y 383.243,Z 345.558,A -85,B 0,C 180,E1 -12153.152,E2 -12153.152} C_VEL
LIN {X 0,Y 383.285,Z 345.555,A -85,B 0,C 180,E1 -12156.315,E2 -12156.315} C_VEL
LIN {X 0,Y 383.249,Z 345.558,A -85,B 0,C 180,E1 -12158.434,E2 -12158.434} C_VEL
LIN {X 0,Y 383.096,Z 345.579,A -85,B 0,C 180,E1 -12161.641,E2 -12161.641} C_VEL
LIN {X 0,Y 383.099,Z 345.575,A -85,B 0,C 180,E1 -12164.881,E2 -12164.881} C_VEL
LIN {X 0,Y 383.05,Z 345.583,A -85,B 0,C 180,E1 -12168.173,E2 -12168.173} C_VEL
LIN {X 0,Y 382.98,Z 345.595,A -85,B 0,C 180,E1 -12171.53,E2 -12171.53} C_VEL
LIN {X 0,Y 383.034,Z 345.584,A -85,B 0,C 180,E1 -12174.911,E2 -12174.911} C_VEL
LIN {X 0,Y 382.416,Z 345.665,A -85,B 0,C 180,E1 -12175.789,E2 -12175.789} C_VEL
LIN {X 0,Y 379.554,Z 346.024,A -85,B 0,C 180,E1 -12177.216,E2 -12177.216} C_VEL
LIN {X 0,Y 377.093,Z 346.327,A -85,B 0,C 180,E1 -12178.37,E2 -12178.37} C_VEL
LIN {X 0,Y 376.028,Z 346.46,A -85,B 0,C 180,E1 -12179.262,E2 -12179.262} C_VEL
LIN {X 0,Y 375.938,Z 346.466,A -85,B 0,C 180,E1 -12179.565,E2 -12179.565} C_VEL
LIN {X 0,Y 375.935,Z 346.469,A -85,B 0,C 180,E1 -12182.828,E2 -12182.828} C_VEL
LIN {X 0,Y 375.944,Z 346.471,A -85,B 0,C 180,E1 -12185.415,E2 -12185.415} C_VEL
LIN {X 0,Y 375.968,Z 346.464,A -85,B 0,C 180,E1 -12188.272,E2 -12188.272} C_VEL
LIN {X 0,Y 375.975,Z 346.465,A -85,B 0,C 180,E1 -12191.61,E2 -12191.61} C_VEL
LIN {X 0,Y 376,Z 346.464,A -85,B 0,C 180,E1 -12195.255,E2 -12195.255} C_VEL
LIN {X 0,Y 375.986,Z 346.465,A -85,B 0,C 180,E1 -12199.141,E2 -12199.141} C_VEL
LIN {X 0,Y 375.953,Z 346.465,A -85,B 0,C 180,E1 -12201.912,E2 -12201.912} C_VEL
LIN {X 0,Y 375.965,Z 346.465,A -85,B 0,C 180,E1 -12205.333,E2 -12205.333} C_VEL
LIN {X 0,Y 375.947,Z 346.47,A -85,B 0,C 180,E1 -12208.439,E2 -12208.439} C_VEL
LIN {X 0,Y 375.988,Z 346.463,A -85,B 0,C 180,E1 -12212.142,E2 -12212.142} C_VEL
LIN {X 0,Y 375.994,Z 346.464,A -85,B 0,C 180,E1 -12214.54,E2 -12214.54} C_VEL
LIN {X 0,Y 376.01,Z 346.461,A -85,B 0,C 180,E1 -12218.05,E2 -12218.05} C_VEL
LIN {X 0,Y 376.019,Z 346.457,A -85,B 0,C 180,E1 -12221.475,E2 -12221.475} C_VEL
LIN {X 0,Y 376.049,Z 346.455,A -85,B 0,C 180,E1 -12224.833,E2 -12224.833} C_VEL
LIN {X 0,Y 376.046,Z 346.458,A -85,B 0,C 180,E1 -12228.138,E2 -12228.138} C_VEL
LIN {X 0,Y 376.245,Z 346.432,A -85,B 0,C 180,E1 -12231.878,E2 -12231.878} C_VEL
LIN {X 0,Y 376.161,Z 346.441,A -85,B 0,C 180,E1 -12234.641,E2 -12234.641} C_VEL
LIN {X 0,Y 376.343,Z 346.421,A -85,B 0,C 180,E1 -12237.861,E2 -12237.861} C_VEL
LIN {X 0,Y 376.477,Z 346.404,A -85,B 0,C 180,E1 -12240.001,E2 -12240.001} C_VEL
LIN {X 0,Y 376.182,Z 346.438,A -85,B 0,C 180,E1 -12243.214,E2 -12243.214} C_VEL
LIN {X 0,Y 376.236,Z 346.431,A -85,B 0,C 180,E1 -12246.436,E2 -12246.436} C_VEL
LIN {X 0,Y 376.196,Z 346.435,A -85,B 0,C 180,E1 -12248.596,E2 -12248.596} C_VEL
LIN {X 0,Y 376.05,Z 346.457,A -85,B 0,C 180,E1 -12251.864,E2 -12251.864} C_VEL
LIN {X 0,Y 376.05,Z 346.455,A -85,B 0,C 180,E1 -12255.169,E2 -12255.169} C_VEL
LIN {X 0,Y 376,Z 346.459,A -85,B 0,C 180,E1 -12258.528,E2 -12258.528} C_VEL
LIN {X 0,Y 375.954,Z 346.467,A -85,B 0,C 180,E1 -12261.956,E2 -12261.956} C_VEL
LIN {X 0,Y 375.998,Z 346.464,A -85,B 0,C 180,E1 -12265.462,E2 -12265.462} C_VEL
LIN {X 0,Y 375.969,Z 346.468,A -85,B 0,C 180,E1 -12269.08,E2 -12269.08} C_VEL
LIN {X 0,Y 375.942,Z 346.47,A -85,B 0,C 180,E1 -12272.83,E2 -12272.83} C_VEL
LIN {X 0,Y 375.951,Z 346.469,A -85,B 0,C 180,E1 -12275.417,E2 -12275.417} C_VEL
LIN {X 0,Y 375.969,Z 346.464,A -85,B 0,C 180,E1 -12278.272,E2 -12278.272} C_VEL
LIN {X 0,Y 375.929,Z 346.469,A -85,B 0,C 180,E1 -12281.602,E2 -12281.602} C_VEL
LIN {X 0,Y 375.95,Z 346.468,A -85,B 0,C 180,E1 -12285.266,E2 -12285.266} C_VEL
LIN {X 0,Y 375.937,Z 346.47,A -85,B 0,C 180,E1 -12289.135,E2 -12289.135} C_VEL
LIN {X 0,Y 376.046,Z 346.621,A -85,B 0,C 180,E1 -12291.167,E2 -12291.167} C_VEL
LIN {X 0,Y 377.132,Z 352.828,A -85,B 0,C 180,E1 -12294.713,E2 -12294.713} C_VEL
LIN {X 0,Y 377.523,Z 356.86,A -85,B 0,C 180,E1 -12296.901,E2 -12296.901} C_VEL
LIN {X 0,Y 376.972,Z 362.486,A -85,B 0,C 180,E1 -12299.779,E2 -12299.779} C_VEL
LIN {X 0,Y 376.314,Z 369.704,A -85,B 0,C 180,E1 -12303.372,E2 -12303.372} C_VEL
LIN {X 0,Y 375.72,Z 376.918,A -85,B 0,C 180,E1 -12306.872,E2 -12306.872} C_VEL
LIN {X 0,Y 375.296,Z 384.163,A -85,B 0,C 180,E1 -12310.303,E2 -12310.303} C_VEL
LIN {X 0,Y 374.955,Z 391.353,A -85,B 0,C 180,E1 -12313.673,E2 -12313.673} C_VEL
LIN {X 0,Y 374.853,Z 394.426,A -85,B 0,C 180,E1 -12315.097,E2 -12315.097} C_VEL
LIN {X 0,Y 376.359,Z 407.925,A -85,B 0,C 180,E1 -12315.745,E2 -12315.745} C_VEL
LIN {X 0,Y 377.168,Z 417.702,A -85,B 0,C 180,E1 -12316.391,E2 -12316.391} C_VEL
LIN {X 0,Y 377.358,Z 424.917,A -85,B 0,C 180,E1 -12316.973,E2 -12316.973} C_VEL
LIN {X 0,Y 376.826,Z 433.009,A -85,B 0,C 180,E1 -12317.753,E2 -12317.753} C_VEL
LIN {X 0,Y 376.303,Z 440.915,A -85,B 0,C 180,E1 -12318.692,E2 -12318.692} C_VEL
LIN {X 0,Y 375.759,Z 448.312,A -85,B 0,C 180,E1 -12319.767,E2 -12319.767} C_VEL
LIN {X 0,Y 375.276,Z 455.827,A -85,B 0,C 180,E1 -12321.114,E2 -12321.114} C_VEL
LIN {X 0,Y 374.9,Z 461.726,A -85,B 0,C 180,E1 -12322.461,E2 -12322.461} C_VEL
LIN {X 0,Y 374.663,Z 466.395,A -85,B 0,C 180,E1 -12323.821,E2 -12323.821} C_VEL
LIN {X 0,Y 374.625,Z 469.965,A -85,B 0,C 180,E1 -12325.159,E2 -12325.159} C_VEL
LIN {X 0,Y 374.526,Z 473.03,A -85,B 0,C 180,E1 -12326.774,E2 -12326.774} C_VEL
LIN {X 0,Y 374.593,Z 474.43,A -85,B 0,C 180,E1 -12327.851,E2 -12327.851} C_VEL
LIN {X 0,Y 374.625,Z 475.329,A -85,B 0,C 180,E1 -12328.926,E2 -12328.926} C_VEL
LIN {X 0,Y 374.607,Z 475.633,A -85,B 0,C 180,E1 -12330.001,E2 -12330.001} C_VEL
LIN {X 0,Y 374.623,Z 475.418,A -85,B 0,C 180,E1 -12331.076,E2 -12331.076} C_VEL
LIN {X 0,Y 374.558,Z 474.729,A -85,B 0,C 180,E1 -12332.152,E2 -12332.152} C_VEL
LIN {X 0,Y 374.514,Z 473.561,A -85,B 0,C 180,E1 -12333.229,E2 -12333.229} C_VEL
LIN {X 0,Y 374.626,Z 470.717,A -85,B 0,C 180,E1 -12334.844,E2 -12334.844} C_VEL
LIN {X 0,Y 374.683,Z 467.338,A -85,B 0,C 180,E1 -12336.208,E2 -12336.208} C_VEL
LIN {X 0,Y 374.924,Z 463.041,A -85,B 0,C 180,E1 -12337.541,E2 -12337.541} C_VEL
LIN {X 0,Y 375.306,Z 457.564,A -85,B 0,C 180,E1 -12338.889,E2 -12338.889} C_VEL
LIN {X 0,Y 375.853,Z 450.758,A -85,B 0,C 180,E1 -12340.234,E2 -12340.234} C_VEL
LIN {X 0,Y 376.555,Z 442.051,A -85,B 0,C 180,E1 -12341.576,E2 -12341.576} C_VEL
LIN {X 0,Y 377.2,Z 434.498,A -85,B 0,C 180,E1 -12342.511,E2 -12342.511} C_VEL
LIN {X 0,Y 377.791,Z 426.65,A -85,B 0,C 180,E1 -12343.311,E2 -12343.311} C_VEL
LIN {X 0,Y 377.772,Z 418.655,A -85,B 0,C 180,E1 -12343.997,E2 -12343.997} C_VEL
LIN {X 0,Y 377.129,Z 409.846,A -85,B 0,C 180,E1 -12344.626,E2 -12344.626} C_VEL
LIN {X 0,Y 375.961,Z 400.26,A -85,B 0,C 180,E1 -12345.173,E2 -12345.173} C_VEL
LIN {X 0,Y 374.91,Z 393.465,A -85,B 0,C 180,E1 -12345.495,E2 -12345.495} C_VEL
LIN {X 0,Y 375.203,Z 386.836,A -85,B 0,C 180,E1 -12348.569,E2 -12348.569} C_VEL
LIN {X 0,Y 375.598,Z 379.667,A -85,B 0,C 180,E1 -12351.978,E2 -12351.978} C_VEL
LIN {X 0,Y 376.149,Z 372.614,A -85,B 0,C 180,E1 -12355.452,E2 -12355.452} C_VEL
LIN {X 0,Y 376.814,Z 365.626,A -85,B 0,C 180,E1 -12359.009,E2 -12359.009} C_VEL
LIN {X 0,Y 377.532,Z 359.915,A -85,B 0,C 180,E1 -12362.044,E2 -12362.044} C_VEL
LIN {X 0,Y 377.659,Z 356.583,A -85,B 0,C 180,E1 -12363.938,E2 -12363.938} C_VEL
LIN {X 0,Y 376.78,Z 351.093,A -85,B 0,C 180,E1 -12367.317,E2 -12367.317} C_VEL
LIN {X 0,Y 376.004,Z 346.47,A -85,B 0,C 180,E1 -12370.496,E2 -12370.496} C_VEL
LIN {X 0,Y 375.937,Z 346.477,A -85,B 0,C 180,E1 -12373.766,E2 -12373.766} C_VEL
LIN {X 0,Y 375.941,Z 346.472,A -85,B 0,C 180,E1 -12376.811,E2 -12376.811} C_VEL
LIN {X 0,Y 375.968,Z 346.467,A -85,B 0,C 180,E1 -12380.537,E2 -12380.537} C_VEL
LIN {X 0,Y 375.97,Z 346.467,A -85,B 0,C 180,E1 -12383.496,E2 -12383.496} C_VEL
LIN {X 0,Y 375.967,Z 346.467,A -85,B 0,C 180,E1 -12385.889,E2 -12385.889} C_VEL
LIN {X 0,Y 375.972,Z 346.466,A -85,B 0,C 180,E1 -12389.687,E2 -12389.687} C_VEL
LIN {X 0,Y 376.028,Z 346.459,A -85,B 0,C 180,E1 -12393.348,E2 -12393.348} C_VEL
LIN {X 0,Y 376.004,Z 346.462,A -85,B 0,C 180,E1 -12396.888,E2 -12396.888} C_VEL
LIN {X 0,Y 376.005,Z 346.462,A -85,B 0,C 180,E1 -12400.339,E2 -12400.339} C_VEL
LIN {X 0,Y 376.036,Z 346.459,A -85,B 0,C 180,E1 -12403.718,E2 -12403.718} C_VEL
LIN {X 0,Y 376.111,Z 346.45,A -85,B 0,C 180,E1 -12407.041,E2 -12407.041} C_VEL
LIN {X 0,Y 376.12,Z 346.448,A -85,B 0,C 180,E1 -12410.318,E2 -12410.318} C_VEL
LIN {X 0,Y 376.219,Z 346.435,A -85,B 0,C 180,E1 -12413.564,E2 -12413.564} C_VEL
LIN {X 0,Y 376.355,Z 346.418,A -85,B 0,C 180,E1 -12417.859,E2 -12417.859} C_VEL
LIN {X 0,Y 376.493,Z 346.403,A -85,B 0,C 180,E1 -12419.999,E2 -12419.999} C_VEL
LIN {X 0,Y 376.188,Z 346.439,A -85,B 0,C 180,E1 -12423.212,E2 -12423.212} C_VEL
LIN {X 0,Y 376.219,Z 346.435,A -85,B 0,C 180,E1 -12426.589,E2 -12426.589} C_VEL
LIN {X 0,Y 376.118,Z 346.449,A -85,B 0,C 180,E1 -12429.68,E2 -12429.68} C_VEL
LIN {X 0,Y 376.094,Z 346.454,A -85,B 0,C 180,E1 -12433.656,E2 -12433.656} C_VEL
LIN {X 0,Y 375.985,Z 346.47,A -85,B 0,C 180,E1 -12436.282,E2 -12436.282} C_VEL
LIN {X 0,Y 375.747,Z 346.496,A -85,B 0,C 180,E1 -12438.539,E2 -12438.539} C_VEL
LIN {X 0,Y 375.628,Z 348.202,A -85,B 0,C 180,E1 -12440.689,E2 -12440.689} C_VEL
LIN {X 0,Y 375.395,Z 351.888,A -85,B 0,C 180,E1 -12444.321,E2 -12444.321} C_VEL
LIN {X 0,Y 375.195,Z 355.65,A -85,B 0,C 180,E1 -12447.922,E2 -12447.922} C_VEL
LIN {X 0,Y 375.029,Z 359.662,A -85,B 0,C 180,E1 -12451.648,E2 -12451.648} C_VEL
LIN {X 0,Y 374.914,Z 362.984,A -85,B 0,C 180,E1 -12454.634,E2 -12454.634} C_VEL
LIN {X 0,Y 377.38,Z 373.726,A -85,B 0,C 180,E1 -12455.26,E2 -12455.26} C_VEL
LIN {X 0,Y 378.987,Z 382.525,A -85,B 0,C 180,E1 -12455.904,E2 -12455.904} C_VEL
LIN {X 0,Y 378.993,Z 387.887,A -85,B 0,C 180,E1 -12456.315,E2 -12456.315} C_VEL
LIN {X 0,Y 378.294,Z 397.908,A -85,B 0,C 180,E1 -12457.262,E2 -12457.262} C_VEL
LIN {X 0,Y 377.631,Z 405.93,A -85,B 0,C 180,E1 -12458.214,E2 -12458.214} C_VEL
LIN {X 0,Y 377.13,Z 412.173,A -85,B 0,C 180,E1 -12459.11,E2 -12459.11} C_VEL
LIN {X 0,Y 376.63,Z 417.89,A -85,B 0,C 180,E1 -12460.085,E2 -12460.085} C_VEL
LIN {X 0,Y 376.102,Z 423.396,A -85,B 0,C 180,E1 -12461.215,E2 -12461.215} C_VEL
LIN {X 0,Y 375.663,Z 427.912,A -85,B 0,C 180,E1 -12462.335,E2 -12462.335} C_VEL
LIN {X 0,Y 375.34,Z 431.819,A -85,B 0,C 180,E1 -12463.527,E2 -12463.527} C_VEL
LIN {X 0,Y 375.079,Z 434.679,A -85,B 0,C 180,E1 -12464.599,E2 -12464.599} C_VEL
LIN {X 0,Y 374.786,Z 437.554,A -85,B 0,C 180,E1 -12466.065,E2 -12466.065} C_VEL
LIN {X 0,Y 374.548,Z 439.416,A -85,B 0,C 180,E1 -12467.505,E2 -12467.505} C_VEL
LIN {X 0,Y 374.474,Z 440.358,A -85,B 0,C 180,E1 -12468.937,E2 -12468.937} C_VEL
LIN {X 0,Y 374.431,Z 440.425,A -85,B 0,C 180,E1 -12470.343,E2 -12470.343} C_VEL
LIN {X 0,Y 374.491,Z 439.388,A -85,B 0,C 180,E1 -12472.016,E2 -12472.016} C_VEL
LIN {X 0,Y 374.708,Z 437.054,A -85,B 0,C 180,E1 -12473.753,E2 -12473.753} C_VEL
LIN {X 0,Y 374.948,Z 433.003,A -85,B 0,C 180,E1 -12475.559,E2 -12475.559} C_VEL
LIN {X 0,Y 375.259,Z 429.289,A -85,B 0,C 180,E1 -12476.782,E2 -12476.782} C_VEL
LIN {X 0,Y 375.716,Z 422.857,A -85,B 0,C 180,E1 -12478.414,E2 -12478.414} C_VEL
LIN {X 0,Y 376.232,Z 416.356,A -85,B 0,C 180,E1 -12479.71,E2 -12479.71} C_VEL
LIN {X 0,Y 376.811,Z 408.267,A -85,B 0,C 180,E1 -12480.991,E2 -12480.991} C_VEL
LIN {X 0,Y 377.37,Z 399.334,A -85,B 0,C 180,E1 -12482.099,E2 -12482.099} C_VEL
LIN {X 0,Y 377.913,Z 391.45,A -85,B 0,C 180,E1 -12482.89,E2 -12482.89} C_VEL
LIN {X 0,Y 378.294,Z 383.772,A -85,B 0,C 180,E1 -12483.519,E2 -12483.519} C_VEL
LIN {X 0,Y 377.772,Z 378.22,A -85,B 0,C 180,E1 -12483.935,E2 -12483.935} C_VEL
LIN {X 0,Y 375.912,Z 367.667,A -85,B 0,C 180,E1 -12484.568,E2 -12484.568} C_VEL
LIN {X 0,Y 374.8,Z 361.891,A -85,B 0,C 180,E1 -12484.859,E2 -12484.859} C_VEL
LIN {X 0,Y 374.823,Z 358.245,A -85,B 0,C 180,E1 -12487.974,E2 -12487.974} C_VEL
LIN {X 0,Y 374.961,Z 354.28,A -85,B 0,C 180,E1 -12491.418,E2 -12491.418} C_VEL
LIN {X 0,Y 375.11,Z 351.704,A -85,B 0,C 180,E1 -12493.677,E2 -12493.677} C_VEL
LIN {X 0,Y 375.306,Z 347.969,A -85,B 0,C 180,E1 -12497.013,E2 -12497.013} C_VEL
LIN {X 0,Y 375.346,Z 346.759,A -85,B 0,C 180,E1 -12498.113,E2 -12498.113} C_VEL
LIN {X 0,Y 375.902,Z 346.472,A -85,B 0,C 180,E1 -12501.397,E2 -12501.397} C_VEL
LIN {X 0,Y 376.183,Z 346.437,A -85,B 0,C 180,E1 -12503.563,E2 -12503.563} C_VEL
LIN {X 0,Y 376.344,Z 346.42,A -85,B 0,C 180,E1 -12507.858,E2 -12507.858} C_VEL
LIN {X 0,Y 376.478,Z 346.404,A -85,B 0,C 180,E1 -12509.999,E2 -12509.999} C_VEL
LIN {X 0,Y 376.182,Z 346.437,A -85,B 0,C 180,E1 -12513.212,E2 -12513.212} C_VEL
LIN {X 0,Y 376.243,Z 346.431,A -85,B 0,C 180,E1 -12516.434,E2 -12516.434} C_VEL
LIN {X 0,Y 376.195,Z 346.436,A -85,B 0,C 180,E1 -12518.594,E2 -12518.594} C_VEL
LIN {X 0,Y 376.048,Z 346.458,A -85,B 0,C 180,E1 -12521.862,E2 -12521.862} C_VEL
LIN {X 0,Y 376.047,Z 346.454,A -85,B 0,C 180,E1 -12525.166,E2 -12525.166} C_VEL
LIN {X 0,Y 375.996,Z 346.46,A -85,B 0,C 180,E1 -12528.526,E2 -12528.526} C_VEL
LIN {X 0,Y 375.949,Z 346.469,A -85,B 0,C 180,E1 -12531.953,E2 -12531.953} C_VEL
LIN {X 0,Y 375.993,Z 346.465,A -85,B 0,C 180,E1 -12535.46,E2 -12535.46} C_VEL
LIN {X 0,Y 375.963,Z 346.467,A -85,B 0,C 180,E1 -12539.078,E2 -12539.078} C_VEL
LIN {X 0,Y 375.938,Z 346.466,A -85,B 0,C 180,E1 -12539.565,E2 -12539.565} C_VEL
LIN {X 0,Y 375.257,Z 346.552,A -85,B 0,C 180,E1 -12540.459,E2 -12540.459} C_VEL
LIN {X 0,Y 372.379,Z 346.912,A -85,B 0,C 180,E1 -12541.913,E2 -12541.913} C_VEL
LIN {X 0,Y 369.964,Z 347.215,A -85,B 0,C 180,E1 -12543.089,E2 -12543.089} C_VEL
LIN {X 0,Y 368.951,Z 347.338,A -85,B 0,C 180,E1 -12543.998,E2 -12543.998} C_VEL
LIN {X 0,Y 368.882,Z 347.346,A -85,B 0,C 180,E1 -12544.306,E2 -12544.306} C_VEL
LIN {X 0,Y 368.911,Z 347.345,A -85,B 0,C 180,E1 -12547.56,E2 -12547.56} C_VEL
LIN {X 0,Y 368.938,Z 347.339,A -85,B 0,C 180,E1 -12550.364,E2 -12550.364} C_VEL
LIN {X 0,Y 368.959,Z 347.337,A -85,B 0,C 180,E1 -12553.631,E2 -12553.631} C_VEL
LIN {X 0,Y 368.936,Z 347.342,A -85,B 0,C 180,E1 -12556.705,E2 -12556.705} C_VEL
LIN {X 0,Y 368.938,Z 347.339,A -85,B 0,C 180,E1 -12559.635,E2 -12559.635} C_VEL
LIN {X 0,Y 368.889,Z 347.348,A -85,B 0,C 180,E1 -12563.144,E2 -12563.144} C_VEL
LIN {X 0,Y 368.882,Z 347.349,A -85,B 0,C 180,E1 -12566.462,E2 -12566.462} C_VEL
LIN {X 0,Y 368.909,Z 347.345,A -85,B 0,C 180,E1 -12570.311,E2 -12570.311} C_VEL
LIN {X 0,Y 368.968,Z 347.335,A -85,B 0,C 180,E1 -12573.536,E2 -12573.536} C_VEL
LIN {X 0,Y 368.972,Z 347.339,A -85,B 0,C 180,E1 -12576.423,E2 -12576.423} C_VEL
LIN {X 0,Y 368.949,Z 347.339,A -85,B 0,C 180,E1 -12579.949,E2 -12579.949} C_VEL
LIN {X 0,Y 368.966,Z 347.336,A -85,B 0,C 180,E1 -12583.4,E2 -12583.4} C_VEL
LIN {X 0,Y 369.047,Z 347.327,A -85,B 0,C 180,E1 -12586.791,E2 -12586.791} C_VEL
LIN {X 0,Y 369.06,Z 347.328,A -85,B 0,C 180,E1 -12590.133,E2 -12590.133} C_VEL
LIN {X 0,Y 369.176,Z 347.313,A -85,B 0,C 180,E1 -12592.343,E2 -12592.343} C_VEL
LIN {X 0,Y 369.133,Z 347.316,A -85,B 0,C 180,E1 -12594.539,E2 -12594.539} C_VEL
LIN {X 0,Y 369.308,Z 347.297,A -85,B 0,C 180,E1 -12597.82,E2 -12597.82} C_VEL
LIN {X 0,Y 369.447,Z 347.28,A -85,B 0,C 180,E1 -12600.001,E2 -12600.001} C_VEL
LIN {X 0,Y 369.309,Z 347.296,A -85,B 0,C 180,E1 -12602.182,E2 -12602.182} C_VEL
LIN {X 0,Y 369.198,Z 347.307,A -85,B 0,C 180,E1 -12606.559,E2 -12606.559} C_VEL
LIN {X 0,Y 369.129,Z 347.315,A -85,B 0,C 180,E1 -12608.762,E2 -12608.762} C_VEL
LIN {X 0,Y 369.004,Z 347.333,A -85,B 0,C 180,E1 -12612.094,E2 -12612.094} C_VEL
LIN {X 0,Y 368.989,Z 347.337,A -85,B 0,C 180,E1 -12615.466,E2 -12615.466} C_VEL
LIN {X 0,Y 368.949,Z 347.339,A -85,B 0,C 180,E1 -12618.895,E2 -12618.895} C_VEL
LIN {X 0,Y 368.923,Z 347.341,A -85,B 0,C 180,E1 -12622.397,E2 -12622.397} C_VEL
LIN {X 0,Y 368.992,Z 347.333,A -85,B 0,C 180,E1 -12625.982,E2 -12625.982} C_VEL
LIN {X 0,Y 368.96,Z 347.338,A -85,B 0,C 180,E1 -12628.815,E2 -12628.815} C_VEL
LIN {X 0,Y 368.892,Z 347.345,A -85,B 0,C 180,E1 -12632.239,E2 -12632.239} C_VEL
LIN {X 0,Y 368.922,Z 347.346,A -85,B 0,C 180,E1 -12635.003,E2 -12635.003} C_VEL
LIN {X 0,Y 368.904,Z 347.346,A -85,B 0,C 180,E1 -12638.642,E2 -12638.642} C_VEL
LIN {X 0,Y 368.876,Z 347.347,A -85,B 0,C 180,E1 -12642.011,E2 -12642.011} C_VEL
LIN {X 0,Y 368.903,Z 347.347,A -85,B 0,C 180,E1 -12645.182,E2 -12645.182} C_VEL
LIN {X 0,Y 368.879,Z 347.347,A -85,B 0,C 180,E1 -12648.179,E2 -12648.179} C_VEL
LIN {X 0,Y 368.974,Z 347.362,A -85,B 0,C 180,E1 -12650.882,E2 -12650.882} C_VEL
LIN {X 0,Y 370.124,Z 353.971,A -85,B 0,C 180,E1 -12654.736,E2 -12654.736} C_VEL
LIN {X 0,Y 370.501,Z 357.39,A -85,B 0,C 180,E1 -12656.628,E2 -12656.628} C_VEL
LIN {X 0,Y 370.069,Z 362.195,A -85,B 0,C 180,E1 -12659.154,E2 -12659.154} C_VEL
LIN {X 0,Y 369.348,Z 369.409,A -85,B 0,C 180,E1 -12662.829,E2 -12662.829} C_VEL
LIN {X 0,Y 368.72,Z 376.591,A -85,B 0,C 180,E1 -12666.407,E2 -12666.407} C_VEL
LIN {X 0,Y 368.373,Z 382.332,A -85,B 0,C 180,E1 -12669.204,E2 -12669.204} C_VEL
LIN {X 0,Y 367.992,Z 389.68,A -85,B 0,C 180,E1 -12672.731,E2 -12672.731} C_VEL
LIN {X 0,Y 367.767,Z 394.135,A -85,B 0,C 180,E1 -12674.839,E2 -12674.839} C_VEL
LIN {X 0,Y 369.213,Z 406.951,A -85,B 0,C 180,E1 -12675.463,E2 -12675.463} C_VEL
LIN {X 0,Y 370.047,Z 416.335,A -85,B 0,C 180,E1 -12676.084,E2 -12676.084} C_VEL
LIN {X 0,Y 370.374,Z 424.322,A -85,B 0,C 180,E1 -12676.734,E2 -12676.734} C_VEL
LIN {X 0,Y 369.89,Z 432.36,A -85,B 0,C 180,E1 -12677.52,E2 -12677.52} C_VEL
LIN {X 0,Y 369.273,Z 440.312,A -85,B 0,C 180,E1 -12678.474,E2 -12678.474} C_VEL
LIN {X 0,Y 368.886,Z 446.049,A -85,B 0,C 180,E1 -12679.296,E2 -12679.296} C_VEL
LIN {X 0,Y 368.396,Z 452.458,A -85,B 0,C 180,E1 -12680.392,E2 -12680.392} C_VEL
LIN {X 0,Y 368.052,Z 457.79,A -85,B 0,C 180,E1 -12681.491,E2 -12681.491} C_VEL
LIN {X 0,Y 367.749,Z 463.199,A -85,B 0,C 180,E1 -12682.866,E2 -12682.866} C_VEL
LIN {X 0,Y 367.552,Z 466.464,A -85,B 0,C 180,E1 -12683.882,E2 -12683.882} C_VEL
LIN {X 0,Y 367.54,Z 470.717,A -85,B 0,C 180,E1 -12685.615,E2 -12685.615} C_VEL
LIN {X 0,Y 367.442,Z 472.646,A -85,B 0,C 180,E1 -12686.712,E2 -12686.712} C_VEL
LIN {X 0,Y 367.493,Z 474.065,A -85,B 0,C 180,E1 -12687.809,E2 -12687.809} C_VEL
LIN {X 0,Y 367.54,Z 474.978,A -85,B 0,C 180,E1 -12688.906,E2 -12688.906} C_VEL
LIN {X 0,Y 367.541,Z 475.289,A -85,B 0,C 180,E1 -12690.001,E2 -12690.001} C_VEL
LIN {X 0,Y 367.537,Z 475.092,A -85,B 0,C 180,E1 -12691.097,E2 -12691.097} C_VEL
LIN {X 0,Y 367.458,Z 474.421,A -85,B 0,C 180,E1 -12692.194,E2 -12692.194} C_VEL
LIN {X 0,Y 367.43,Z 473.271,A -85,B 0,C 180,E1 -12693.291,E2 -12693.291} C_VEL
LIN {X 0,Y 367.54,Z 471.581,A -85,B 0,C 180,E1 -12694.388,E2 -12694.388} C_VEL
LIN {X 0,Y 367.564,Z 467.625,A -85,B 0,C 180,E1 -12696.136,E2 -12696.136} C_VEL
LIN {X 0,Y 367.785,Z 464.746,A -85,B 0,C 180,E1 -12697.136,E2 -12697.136} C_VEL
LIN {X 0,Y 368.107,Z 459.747,A -85,B 0,C 180,E1 -12698.51,E2 -12698.51} C_VEL
LIN {X 0,Y 368.577,Z 453.465,A -85,B 0,C 180,E1 -12699.883,E2 -12699.883} C_VEL
LIN {X 0,Y 369.135,Z 447.355,A -85,B 0,C 180,E1 -12700.977,E2 -12700.977} C_VEL
LIN {X 0,Y 369.737,Z 439.95,A -85,B 0,C 180,E1 -12702.07,E2 -12702.07} C_VEL
LIN {X 0,Y 370.456,Z 432.057,A -85,B 0,C 180,E1 -12703.021,E2 -12703.021} C_VEL
LIN {X 0,Y 370.956,Z 423.767,A -85,B 0,C 180,E1 -12703.84,E2 -12703.84} C_VEL
LIN {X 0,Y 370.538,Z 413.462,A -85,B 0,C 180,E1 -12704.687,E2 -12704.687} C_VEL
LIN {X 0,Y 369.188,Z 401.613,A -85,B 0,C 180,E1 -12705.425,E2 -12705.425} C_VEL
LIN {X 0,Y 367.879,Z 393.052,A -85,B 0,C 180,E1 -12705.87,E2 -12705.87} C_VEL
LIN {X 0,Y 368.242,Z 385.428,A -85,B 0,C 180,E1 -12709.513,E2 -12709.513} C_VEL
LIN {X 0,Y 368.695,Z 378.323,A -85,B 0,C 180,E1 -12713.004,E2 -12713.004} C_VEL
LIN {X 0,Y 369.307,Z 371.299,A -85,B 0,C 180,E1 -12716.565,E2 -12716.565} C_VEL
LIN {X 0,Y 370.078,Z 364.385,A -85,B 0,C 180,E1 -12720.217,E2 -12720.217} C_VEL
LIN {X 0,Y 370.615,Z 359.895,A -85,B 0,C 180,E1 -12722.715,E2 -12722.715} C_VEL
LIN {X 0,Y 370.466,Z 356.542,A -85,B 0,C 180,E1 -12724.69,E2 -12724.69} C_VEL
LIN {X 0,Y 369.771,Z 352.205,A -85,B 0,C 180,E1 -12727.461,E2 -12727.461} C_VEL
LIN {X 0,Y 368.96,Z 347.348,A -85,B 0,C 180,E1 -12730.813,E2 -12730.813} C_VEL
LIN {X 0,Y 368.887,Z 347.355,A -85,B 0,C 180,E1 -12734.825,E2 -12734.825} C_VEL
LIN {X 0,Y 368.89,Z 347.349,A -85,B 0,C 180,E1 -12738.178,E2 -12738.178} C_VEL
LIN {X 0,Y 368.913,Z 347.347,A -85,B 0,C 180,E1 -12741.36,E2 -12741.36} C_VEL
LIN {X 0,Y 368.944,Z 347.342,A -85,B 0,C 180,E1 -12745.146,E2 -12745.146} C_VEL
LIN {X 0,Y 368.937,Z 347.343,A -85,B 0,C 180,E1 -12749.046,E2 -12749.046} C_VEL
LIN {X 0,Y 368.971,Z 347.339,A -85,B 0,C 180,E1 -12752.796,E2 -12752.796} C_VEL
LIN {X 0,Y 368.953,Z 347.341,A -85,B 0,C 180,E1 -12756.113,E2 -12756.113} C_VEL
LIN {X 0,Y 368.944,Z 347.342,A -85,B 0,C 180,E1 -12759.947,E2 -12759.947} C_VEL
LIN {X 0,Y 368.983,Z 347.337,A -85,B 0,C 180,E1 -12763.398,E2 -12763.398} C_VEL
LIN {X 0,Y 369.065,Z 347.327,A -85,B 0,C 180,E1 -12766.79,E2 -12766.79} C_VEL
LIN {X 0,Y 369.07,Z 347.326,A -85,B 0,C 180,E1 -12770.131,E2 -12770.131} C_VEL
LIN {X 0,Y 369.179,Z 347.312,A -85,B 0,C 180,E1 -12773.44,E2 -12773.44} C_VEL
LIN {X 0,Y 369.32,Z 347.294,A -85,B 0,C 180,E1 -12777.818,E2 -12777.818} C_VEL
LIN {X 0,Y 369.462,Z 347.279,A -85,B 0,C 180,E1 -12779.999,E2 -12779.999} C_VEL
LIN {X 0,Y 369.321,Z 347.295,A -85,B 0,C 180,E1 -12782.18,E2 -12782.18} C_VEL
LIN {X 0,Y 369.192,Z 347.311,A -85,B 0,C 180,E1 -12786.572,E2 -12786.572} C_VEL
LIN {X 0,Y 369.068,Z 347.327,A -85,B 0,C 180,E1 -12789.867,E2 -12789.867} C_VEL
LIN {X 0,Y 369.041,Z 347.332,A -85,B 0,C 180,E1 -12793.771,E2 -12793.771} C_VEL
LIN {X 0,Y 368.909,Z 347.352,A -85,B 0,C 180,E1 -12796.603,E2 -12796.603} C_VEL
LIN {X 0,Y 368.64,Z 347.474,A -85,B 0,C 180,E1 -12798.91,E2 -12798.91} C_VEL
LIN {X 0,Y 368.486,Z 350.893,A -85,B 0,C 180,E1 -12802.422,E2 -12802.422} C_VEL
LIN {X 0,Y 368.252,Z 354.762,A -85,B 0,C 180,E1 -12806.234,E2 -12806.234} C_VEL
LIN {X 0,Y 368.053,Z 358.445,A -85,B 0,C 180,E1 -12809.765,E2 -12809.765} C_VEL
LIN {X 0,Y 367.92,Z 361.706,A -85,B 0,C 180,E1 -12812.807,E2 -12812.807} C_VEL
LIN {X 0,Y 367.851,Z 363.28,A -85,B 0,C 180,E1 -12814.263,E2 -12814.263} C_VEL
LIN {X 0,Y 370.669,Z 375.448,A -85,B 0,C 180,E1 -12815.029,E2 -12815.029} C_VEL
LIN {X 0,Y 372.229,Z 384.381,A -85,B 0,C 180,E1 -12815.719,E2 -12815.719} C_VEL
LIN {X 0,Y 371.909,Z 392.008,A -85,B 0,C 180,E1 -12816.361,E2 -12816.361} C_VEL
LIN {X 0,Y 371.366,Z 399.296,A -85,B 0,C 180,E1 -12817.099,E2 -12817.099} C_VEL
LIN {X 0,Y 370.704,Z 406.882,A -85,B 0,C 180,E1 -12818.033,E2 -12818.033} C_VEL
LIN {X 0,Y 370.034,Z 414.419,A -85,B 0,C 180,E1 -12819.172,E2 -12819.172} C_VEL
LIN {X 0,Y 369.389,Z 421.236,A -85,B 0,C 180,E1 -12820.442,E2 -12820.442} C_VEL
LIN {X 0,Y 368.744,Z 427.686,A -85,B 0,C 180,E1 -12821.984,E2 -12821.984} C_VEL
LIN {X 0,Y 368.286,Z 432.575,A -85,B 0,C 180,E1 -12823.517,E2 -12823.517} C_VEL
LIN {X 0,Y 368.094,Z 434.615,A -85,B 0,C 180,E1 -12824.275,E2 -12824.275} C_VEL
LIN {X 0,Y 367.764,Z 437.631,A -85,B 0,C 180,E1 -12825.77,E2 -12825.77} C_VEL
LIN {X 0,Y 367.612,Z 438.813,A -85,B 0,C 180,E1 -12826.59,E2 -12826.59} C_VEL
LIN {X 0,Y 367.4,Z 440.449,A -85,B 0,C 180,E1 -12828.245,E2 -12828.245} C_VEL
LIN {X 0,Y 367.325,Z 440.884,A -85,B 0,C 180,E1 -12829.933,E2 -12829.933} C_VEL
LIN {X 0,Y 367.369,Z 440.051,A -85,B 0,C 180,E1 -12831.659,E2 -12831.659} C_VEL
LIN {X 0,Y 367.615,Z 437.593,A -85,B 0,C 180,E1 -12833.653,E2 -12833.653} C_VEL
LIN {X 0,Y 367.831,Z 434.378,A -85,B 0,C 180,E1 -12835.241,E2 -12835.241} C_VEL
LIN {X 0,Y 368.186,Z 429.923,A -85,B 0,C 180,E1 -12836.79,E2 -12836.79} C_VEL
LIN {X 0,Y 368.492,Z 425.324,A -85,B 0,C 180,E1 -12838.044,E2 -12838.044} C_VEL
LIN {X 0,Y 368.993,Z 419.244,A -85,B 0,C 180,E1 -12839.369,E2 -12839.369} C_VEL
LIN {X 0,Y 369.52,Z 412.678,A -85,B 0,C 180,E1 -12840.532,E2 -12840.532} C_VEL
LIN {X 0,Y 370.02,Z 404.973,A -85,B 0,C 180,E1 -12841.65,E2 -12841.65} C_VEL
LIN {X 0,Y 370.734,Z 395.195,A -85,B 0,C 180,E1 -12842.783,E2 -12842.783} C_VEL
LIN {X 0,Y 371.299,Z 385.149,A -85,B 0,C 180,E1 -12843.663,E2 -12843.663} C_VEL
LIN {X 0,Y 371.042,Z 380.521,A -85,B 0,C 180,E1 -12844.021,E2 -12844.021} C_VEL
LIN {X 0,Y 369.003,Z 368.777,A -85,B 0,C 180,E1 -12844.775,E2 -12844.775} C_VEL
LIN {X 0,Y 367.743,Z 362.165,A -85,B 0,C 180,E1 -12845.136,E2 -12845.136} C_VEL
LIN {X 0,Y 367.747,Z 358.047,A -85,B 0,C 180,E1 -12848.708,E2 -12848.708} C_VEL
LIN {X 0,Y 368.024,Z 353.5,A -85,B 0,C 180,E1 -12852.707,E2 -12852.707} C_VEL
LIN {X 0,Y 368.227,Z 349.018,A -85,B 0,C 180,E1 -12856.759,E2 -12856.759} C_VEL
LIN {X 0,Y 368.275,Z 347.797,A -85,B 0,C 180,E1 -12857.881,E2 -12857.881} C_VEL
LIN {X 0,Y 368.6,Z 347.385,A -85,B 0,C 180,E1 -12860.118,E2 -12860.118} C_VEL
LIN {X 0,Y 369.025,Z 347.333,A -85,B 0,C 180,E1 -12862.338,E2 -12862.338} C_VEL
LIN {X 0,Y 369.121,Z 347.319,A -85,B 0,C 180,E1 -12864.536,E2 -12864.536} C_VEL
LIN {X 0,Y 369.309,Z 347.296,A -85,B 0,C 180,E1 -12867.817,E2 -12867.817} C_VEL
LIN {X 0,Y 369.448,Z 347.28,A -85,B 0,C 180,E1 -12869.999,E2 -12869.999} C_VEL
LIN {X 0,Y 369.309,Z 347.297,A -85,B 0,C 180,E1 -12872.18,E2 -12872.18} C_VEL
LIN {X 0,Y 369.204,Z 347.307,A -85,B 0,C 180,E1 -12876.557,E2 -12876.557} C_VEL
LIN {X 0,Y 369.127,Z 347.315,A -85,B 0,C 180,E1 -12878.76,E2 -12878.76} C_VEL
LIN {X 0,Y 369.002,Z 347.335,A -85,B 0,C 180,E1 -12882.092,E2 -12882.092} C_VEL
LIN {X 0,Y 368.986,Z 347.336,A -85,B 0,C 180,E1 -12885.464,E2 -12885.464} C_VEL
LIN {X 0,Y 368.945,Z 347.338,A -85,B 0,C 180,E1 -12888.893,E2 -12888.893} C_VEL
LIN {X 0,Y 368.919,Z 347.342,A -85,B 0,C 180,E1 -12892.394,E2 -12892.394} C_VEL
LIN {X 0,Y 368.986,Z 347.335,A -85,B 0,C 180,E1 -12895.979,E2 -12895.979} C_VEL
LIN {X 0,Y 368.91,Z 347.345,A -85,B 0,C 180,E1 -12899.562,E2 -12899.562} C_VEL
LIN {X 0,Y 368.883,Z 347.349,A -85,B 0,C 180,E1 -12903.043,E2 -12903.043} C_VEL
LIN {X 0,Y 368.882,Z 347.346,A -85,B 0,C 180,E1 -12904.306,E2 -12904.306} C_VEL
LIN {X 0,Y 368.252,Z 347.429,A -85,B 0,C 180,E1 -12905.217,E2 -12905.217} C_VEL
LIN {X 0,Y 365.423,Z 347.785,A -85,B 0,C 180,E1 -12906.7,E2 -12906.7} C_VEL
LIN {X 0,Y 362.999,Z 348.088,A -85,B 0,C 180,E1 -12907.899,E2 -12907.899} C_VEL
LIN {X 0,Y 361.949,Z 348.215,A -85,B 0,C 180,E1 -12908.826,E2 -12908.826} C_VEL
LIN {X 0,Y 361.859,Z 348.224,A -85,B 0,C 180,E1 -12909.14,E2 -12909.14} C_VEL
LIN {X 0,Y 361.872,Z 348.22,A -85,B 0,C 180,E1 -12912.44,E2 -12912.44} C_VEL
LIN {X 0,Y 361.914,Z 348.214,A -85,B 0,C 180,E1 -12915.928,E2 -12915.928} C_VEL
LIN {X 0,Y 361.89,Z 348.22,A -85,B 0,C 180,E1 -12919.232,E2 -12919.232} C_VEL
LIN {X 0,Y 361.859,Z 348.225,A -85,B 0,C 180,E1 -12922.983,E2 -12922.983} C_VEL
LIN {X 0,Y 361.844,Z 348.227,A -85,B 0,C 180,E1 -12926.631,E2 -12926.631} C_VEL
LIN {X 0,Y 361.862,Z 348.22,A -85,B 0,C 180,E1 -12929.673,E2 -12929.673} C_VEL
LIN {X 0,Y 361.941,Z 348.21,A -85,B 0,C 180,E1 -12933.476,E2 -12933.476} C_VEL
LIN {X 0,Y 361.908,Z 348.215,A -85,B 0,C 180,E1 -12937.147,E2 -12937.147} C_VEL
LIN {X 0,Y 361.922,Z 348.216,A -85,B 0,C 180,E1 -12940.726,E2 -12940.726} C_VEL
LIN {X 0,Y 361.936,Z 348.216,A -85,B 0,C 180,E1 -12944.227,E2 -12944.227} C_VEL
LIN {X 0,Y 361.987,Z 348.208,A -85,B 0,C 180,E1 -12946.529,E2 -12946.529} C_VEL
LIN {X 0,Y 362.023,Z 348.203,A -85,B 0,C 180,E1 -12949.939,E2 -12949.939} C_VEL
LIN {X 0,Y 362.139,Z 348.191,A -85,B 0,C 180,E1 -12952.194,E2 -12952.194} C_VEL
LIN {X 0,Y 362.107,Z 348.192,A -85,B 0,C 180,E1 -12954.432,E2 -12954.432} C_VEL
LIN {X 0,Y 362.272,Z 348.173,A -85,B 0,C 180,E1 -12957.778,E2 -12957.778} C_VEL
LIN {X 0,Y 362.416,Z 348.156,A -85,B 0,C 180,E1 -12960.001,E2 -12960.001} C_VEL
LIN {X 0,Y 362.273,Z 348.172,A -85,B 0,C 180,E1 -12962.225,E2 -12962.225} C_VEL
LIN {X 0,Y 362.162,Z 348.183,A -85,B 0,C 180,E1 -12966.687,E2 -12966.687} C_VEL
LIN {X 0,Y 362.065,Z 348.195,A -85,B 0,C 180,E1 -12968.934,E2 -12968.934} C_VEL
LIN {X 0,Y 361.957,Z 348.209,A -85,B 0,C 180,E1 -12972.333,E2 -12972.333} C_VEL
LIN {X 0,Y 361.953,Z 348.209,A -85,B 0,C 180,E1 -12974.622,E2 -12974.622} C_VEL
LIN {X 0,Y 361.947,Z 348.211,A -85,B 0,C 180,E1 -12978.101,E2 -12978.101} C_VEL
LIN {X 0,Y 361.883,Z 348.221,A -85,B 0,C 180,E1 -12981.654,E2 -12981.654} C_VEL
LIN {X 0,Y 361.92,Z 348.218,A -85,B 0,C 180,E1 -12985.292,E2 -12985.292} C_VEL
LIN {X 0,Y 361.915,Z 348.215,A -85,B 0,C 180,E1 -12987.779,E2 -12987.779} C_VEL
LIN {X 0,Y 361.84,Z 348.227,A -85,B 0,C 180,E1 -12991.287,E2 -12991.287} C_VEL
LIN {X 0,Y 361.847,Z 348.222,A -85,B 0,C 180,E1 -12994.282,E2 -12994.282} C_VEL
LIN {X 0,Y 361.858,Z 348.225,A -85,B 0,C 180,E1 -12997.225,E2 -12997.225} C_VEL
LIN {X 0,Y 361.83,Z 348.228,A -85,B 0,C 180,E1 -13000.757,E2 -13000.757} C_VEL
LIN {X 0,Y 361.83,Z 348.226,A -85,B 0,C 180,E1 -13004.367,E2 -13004.367} C_VEL
LIN {X 0,Y 361.832,Z 348.224,A -85,B 0,C 180,E1 -13007.57,E2 -13007.57} C_VEL
LIN {X 0,Y 361.929,Z 348.302,A -85,B 0,C 180,E1 -13010.711,E2 -13010.711} C_VEL
LIN {X 0,Y 362.809,Z 353.435,A -85,B 0,C 180,E1 -13013.788,E2 -13013.788} C_VEL
LIN {X 0,Y 363.428,Z 357.741,A -85,B 0,C 180,E1 -13016.258,E2 -13016.258} C_VEL
LIN {X 0,Y 363.172,Z 361.891,A -85,B 0,C 180,E1 -13018.502,E2 -13018.502} C_VEL
LIN {X 0,Y 362.392,Z 369.075,A -85,B 0,C 180,E1 -13022.263,E2 -13022.263} C_VEL
LIN {X 0,Y 361.75,Z 376.284,A -85,B 0,C 180,E1 -13025.939,E2 -13025.939} C_VEL
LIN {X 0,Y 361.224,Z 383.453,A -85,B 0,C 180,E1 -13029.502,E2 -13029.502} C_VEL
LIN {X 0,Y 360.873,Z 390.599,A -85,B 0,C 180,E1 -13033.016,E2 -13033.016} C_VEL
LIN {X 0,Y 360.682,Z 393.873,A -85,B 0,C 180,E1 -13034.606,E2 -13034.606} C_VEL
LIN {X 0,Y 362.074,Z 405.894,A -85,B 0,C 180,E1 -13035.17,E2 -13035.17} C_VEL
LIN {X 0,Y 362.944,Z 415.464,A -85,B 0,C 180,E1 -13035.806,E2 -13035.806} C_VEL
LIN {X 0,Y 363.352,Z 424.709,A -85,B 0,C 180,E1 -13036.581,E2 -13036.581} C_VEL
LIN {X 0,Y 362.962,Z 431.704,A -85,B 0,C 180,E1 -13037.278,E2 -13037.278} C_VEL
LIN {X 0,Y 362.296,Z 439.709,A -85,B 0,C 180,E1 -13038.249,E2 -13038.249} C_VEL
LIN {X 0,Y 361.897,Z 445.493,A -85,B 0,C 180,E1 -13039.087,E2 -13039.087} C_VEL
LIN {X 0,Y 361.363,Z 451.94,A -85,B 0,C 180,E1 -13040.204,E2 -13040.204} C_VEL
LIN {X 0,Y 361.017,Z 457.306,A -85,B 0,C 180,E1 -13041.324,E2 -13041.324} C_VEL
LIN {X 0,Y 360.689,Z 462.742,A -85,B 0,C 180,E1 -13042.725,E2 -13042.725} C_VEL
LIN {X 0,Y 360.448,Z 466.506,A -85,B 0,C 180,E1 -13043.934,E2 -13043.934} C_VEL
LIN {X 0,Y 360.447,Z 470.31,A -85,B 0,C 180,E1 -13045.528,E2 -13045.528} C_VEL
LIN {X 0,Y 360.36,Z 472.262,A -85,B 0,C 180,E1 -13046.647,E2 -13046.647} C_VEL
LIN {X 0,Y 360.394,Z 473.701,A -85,B 0,C 180,E1 -13047.766,E2 -13047.766} C_VEL
LIN {X 0,Y 360.458,Z 474.625,A -85,B 0,C 180,E1 -13048.884,E2 -13048.884} C_VEL
LIN {X 0,Y 360.477,Z 474.945,A -85,B 0,C 180,E1 -13050.001,E2 -13050.001} C_VEL
LIN {X 0,Y 360.454,Z 474.766,A -85,B 0,C 180,E1 -13051.119,E2 -13051.119} C_VEL
LIN {X 0,Y 360.359,Z 474.114,A -85,B 0,C 180,E1 -13052.237,E2 -13052.237} C_VEL
LIN {X 0,Y 360.35,Z 472.988,A -85,B 0,C 180,E1 -13053.356,E2 -13053.356} C_VEL
LIN {X 0,Y 360.428,Z 470.183,A -85,B 0,C 180,E1 -13055.035,E2 -13055.035} C_VEL
LIN {X 0,Y 360.459,Z 467.878,A -85,B 0,C 180,E1 -13056.082,E2 -13056.082} C_VEL
LIN {X 0,Y 360.717,Z 464.534,A -85,B 0,C 180,E1 -13057.277,E2 -13057.277} C_VEL
LIN {X 0,Y 361.148,Z 458.389,A -85,B 0,C 180,E1 -13058.958,E2 -13058.958} C_VEL
LIN {X 0,Y 361.581,Z 453.33,A -85,B 0,C 180,E1 -13060.076,E2 -13060.076} C_VEL
LIN {X 0,Y 362.161,Z 447.26,A -85,B 0,C 180,E1 -13061.191,E2 -13061.191} C_VEL
LIN {X 0,Y 362.788,Z 439.902,A -85,B 0,C 180,E1 -13062.305,E2 -13062.305} C_VEL
LIN {X 0,Y 363.549,Z 432.069,A -85,B 0,C 180,E1 -13063.273,E2 -13063.273} C_VEL
LIN {X 0,Y 364.055,Z 425.344,A -85,B 0,C 180,E1 -13063.965,E2 -13063.965} C_VEL
LIN {X 0,Y 363.792,Z 416.734,A -85,B 0,C 180,E1 -13064.727,E2 -13064.727} C_VEL
LIN {X 0,Y 363.018,Z 407.794,A -85,B 0,C 180,E1 -13065.379,E2 -13065.379} C_VEL
LIN {X 0,Y 361.502,Z 396.948,A -85,B 0,C 180,E1 -13066.012,E2 -13066.012} C_VEL
LIN {X 0,Y 360.819,Z 392.719,A -85,B 0,C 180,E1 -13066.225,E2 -13066.225} C_VEL
LIN {X 0,Y 361.223,Z 385.218,A -85,B 0,C 180,E1 -13069.908,E2 -13069.908} C_VEL
LIN {X 0,Y 361.698,Z 378.137,A -85,B 0,C 180,E1 -13073.475,E2 -13073.475} C_VEL
LIN {X 0,Y 362.303,Z 371.709,A -85,B 0,C 180,E1 -13076.833,E2 -13076.833} C_VEL
LIN {X 0,Y 363.195,Z 364.316,A -85,B 0,C 180,E1 -13080.851,E2 -13080.851} C_VEL
LIN {X 0,Y 363.609,Z 360.942,A -85,B 0,C 180,E1 -13082.766,E2 -13082.766} C_VEL
LIN {X 0,Y 363.473,Z 357.638,A -85,B 0,C 180,E1 -13084.78,E2 -13084.78} C_VEL
LIN {X 0,Y 362.586,Z 352.246,A -85,B 0,C 180,E1 -13088.336,E2 -13088.336} C_VEL
LIN {X 0,Y 361.887,Z 348.229,A -85,B 0,C 180,E1 -13091.324,E2 -13091.324} C_VEL
LIN {X 0,Y 361.824,Z 348.234,A -85,B 0,C 180,E1 -13094.369,E2 -13094.369} C_VEL
LIN {X 0,Y 361.843,Z 348.228,A -85,B 0,C 180,E1 -13097.568,E2 -13097.568} C_VEL
LIN {X 0,Y 361.875,Z 348.223,A -85,B 0,C 180,E1 -13100.974,E2 -13100.974} C_VEL
LIN {X 0,Y 361.882,Z 348.222,A -85,B 0,C 180,E1 -13104.655,E2 -13104.655} C_VEL
LIN {X 0,Y 361.845,Z 348.226,A -85,B 0,C 180,E1 -13108.37,E2 -13108.37} C_VEL
LIN {X 0,Y 361.916,Z 348.217,A -85,B 0,C 180,E1 -13112.221,E2 -13112.221} C_VEL
LIN {X 0,Y 361.936,Z 348.215,A -85,B 0,C 180,E1 -13114.71,E2 -13114.71} C_VEL
LIN {X 0,Y 361.9,Z 348.218,A -85,B 0,C 180,E1 -13118.347,E2 -13118.347} C_VEL
LIN {X 0,Y 361.975,Z 348.21,A -85,B 0,C 180,E1 -13122.061,E2 -13122.061} C_VEL
LIN {X 0,Y 362.005,Z 348.206,A -85,B 0,C 180,E1 -13126.101,E2 -13126.101} C_VEL
LIN {X 0,Y 362.007,Z 348.206,A -85,B 0,C 180,E1 -13129.936,E2 -13129.936} C_VEL
LIN {X 0,Y 362.142,Z 348.189,A -85,B 0,C 180,E1 -13133.312,E2 -13133.312} C_VEL
LIN {X 0,Y 362.283,Z 348.171,A -85,B 0,C 180,E1 -13137.775,E2 -13137.775} C_VEL
LIN {X 0,Y 362.432,Z 348.154,A -85,B 0,C 180,E1 -13139.999,E2 -13139.999} C_VEL
LIN {X 0,Y 362.285,Z 348.172,A -85,B 0,C 180,E1 -13142.222,E2 -13142.222} C_VEL
LIN {X 0,Y 362.154,Z 348.188,A -85,B 0,C 180,E1 -13146.685,E2 -13146.685} C_VEL
LIN {X 0,Y 362.004,Z 348.206,A -85,B 0,C 180,E1 -13150.062,E2 -13150.062} C_VEL
LIN {X 0,Y 361.999,Z 348.21,A -85,B 0,C 180,E1 -13153.895,E2 -13153.895} C_VEL
LIN {X 0,Y 361.839,Z 348.231,A -85,B 0,C 180,E1 -13156.937,E2 -13156.937} C_VEL
LIN {X 0,Y 361.713,Z 348.245,A -85,B 0,C 180,E1 -13158.111,E2 -13158.111} C_VEL
LIN {X 0,Y 361.594,Z 348.853,A -85,B 0,C 180,E1 -13159.293,E2 -13159.293} C_VEL
LIN {X 0,Y 361.479,Z 351.144,A -85,B 0,C 180,E1 -13161.677,E2 -13161.677} C_VEL
LIN {X 0,Y 361.263,Z 354.745,A -85,B 0,C 180,E1 -13165.338,E2 -13165.338} C_VEL
LIN {X 0,Y 361.03,Z 358.593,A -85,B 0,C 180,E1 -13169.12,E2 -13169.12} C_VEL
LIN {X 0,Y 360.891,Z 361.323,A -85,B 0,C 180,E1 -13171.72,E2 -13171.72} C_VEL
LIN {X 0,Y 360.809,Z 363.631,A -85,B 0,C 180,E1 -13173.886,E2 -13173.886} C_VEL
LIN {X 0,Y 363.514,Z 374.955,A -85,B 0,C 180,E1 -13174.622,E2 -13174.622} C_VEL
LIN {X 0,Y 365.078,Z 383.327,A -85,B 0,C 180,E1 -13175.274,E2 -13175.274} C_VEL
LIN {X 0,Y 365.47,Z 387.005,A -85,B 0,C 180,E1 -13175.587,E2 -13175.587} C_VEL
LIN {X 0,Y 364.779,Z 396.771,A -85,B 0,C 180,E1 -13176.485,E2 -13176.485} C_VEL
LIN {X 0,Y 363.865,Z 406.319,A -85,B 0,C 180,E1 -13177.634,E2 -13177.634} C_VEL
LIN {X 0,Y 363.247,Z 413.532,A -85,B 0,C 180,E1 -13178.718,E2 -13178.718} C_VEL
LIN {X 0,Y 362.687,Z 419.238,A -85,B 0,C 180,E1 -13179.75,E2 -13179.75} C_VEL
LIN {X 0,Y 362.092,Z 425.026,A -85,B 0,C 180,E1 -13181.018,E2 -13181.018} C_VEL
LIN {X 0,Y 361.51,Z 430.019,A -85,B 0,C 180,E1 -13182.374,E2 -13182.374} C_VEL
LIN {X 0,Y 361.086,Z 434.48,A -85,B 0,C 180,E1 -13183.932,E2 -13183.932} C_VEL
LIN {X 0,Y 360.741,Z 437.68,A -85,B 0,C 180,E1 -13185.463,E2 -13185.463} C_VEL
LIN {X 0,Y 360.474,Z 439.788,A -85,B 0,C 180,E1 -13186.969,E2 -13186.969} C_VEL
LIN {X 0,Y 360.291,Z 440.941,A -85,B 0,C 180,E1 -13188.453,E2 -13188.453} C_VEL
LIN {X 0,Y 360.248,Z 441.211,A -85,B 0,C 180,E1 -13189.924,E2 -13189.924} C_VEL
LIN {X 0,Y 360.263,Z 440.634,A -85,B 0,C 180,E1 -13191.371,E2 -13191.371} C_VEL
LIN {X 0,Y 360.412,Z 438.821,A -85,B 0,C 180,E1 -13193.079,E2 -13193.079} C_VEL
LIN {X 0,Y 360.603,Z 436.99,A -85,B 0,C 180,E1 -13194.218,E2 -13194.218} C_VEL
LIN {X 0,Y 360.808,Z 433.917,A -85,B 0,C 180,E1 -13195.605,E2 -13195.605} C_VEL
LIN {X 0,Y 361.14,Z 429.906,A -85,B 0,C 180,E1 -13196.981,E2 -13196.981} C_VEL
LIN {X 0,Y 361.51,Z 424.894,A -85,B 0,C 180,E1 -13198.337,E2 -13198.337} C_VEL
LIN {X 0,Y 361.937,Z 419.85,A -85,B 0,C 180,E1 -13199.454,E2 -13199.454} C_VEL
LIN {X 0,Y 362.431,Z 413.938,A -85,B 0,C 180,E1 -13200.542,E2 -13200.542} C_VEL
LIN {X 0,Y 362.953,Z 406.434,A -85,B 0,C 180,E1 -13201.678,E2 -13201.678} C_VEL
LIN {X 0,Y 363.52,Z 399.052,A -85,B 0,C 180,E1 -13202.594,E2 -13202.594} C_VEL
LIN {X 0,Y 364.115,Z 390.037,A -85,B 0,C 180,E1 -13203.502,E2 -13203.502} C_VEL
LIN {X 0,Y 364.254,Z 382.506,A -85,B 0,C 180,E1 -13204.116,E2 -13204.116} C_VEL
LIN {X 0,Y 362.403,Z 371.399,A -85,B 0,C 180,E1 -13204.898,E2 -13204.898} C_VEL
LIN {X 0,Y 360.674,Z 362.482,A -85,B 0,C 180,E1 -13205.384,E2 -13205.384} C_VEL
LIN {X 0,Y 360.747,Z 357.832,A -85,B 0,C 180,E1 -13209.47,E2 -13209.47} C_VEL
LIN {X 0,Y 360.96,Z 353.87,A -85,B 0,C 180,E1 -13213.018,E2 -13213.018} C_VEL
LIN {X 0,Y 361.146,Z 349.897,A -85,B 0,C 180,E1 -13216.651,E2 -13216.651} C_VEL
LIN {X 0,Y 361.212,Z 348.831,A -85,B 0,C 180,E1 -13217.64,E2 -13217.64} C_VEL
LIN {X 0,Y 361.335,Z 348.29,A -85,B 0,C 180,E1 -13218.783,E2 -13218.783} C_VEL
LIN {X 0,Y 361.969,Z 348.212,A -85,B 0,C 180,E1 -13222.187,E2 -13222.187} C_VEL
LIN {X 0,Y 362.09,Z 348.196,A -85,B 0,C 180,E1 -13224.429,E2 -13224.429} C_VEL
LIN {X 0,Y 362.273,Z 348.172,A -85,B 0,C 180,E1 -13227.775,E2 -13227.775} C_VEL
LIN {X 0,Y 362.418,Z 348.156,A -85,B 0,C 180,E1 -13229.999,E2 -13229.999} C_VEL
LIN {X 0,Y 362.273,Z 348.173,A -85,B 0,C 180,E1 -13232.222,E2 -13232.222} C_VEL
LIN {X 0,Y 362.166,Z 348.183,A -85,B 0,C 180,E1 -13236.685,E2 -13236.685} C_VEL
LIN {X 0,Y 362.064,Z 348.195,A -85,B 0,C 180,E1 -13238.932,E2 -13238.932} C_VEL
LIN {X 0,Y 361.955,Z 348.21,A -85,B 0,C 180,E1 -13242.331,E2 -13242.331} C_VEL
LIN {X 0,Y 361.95,Z 348.209,A -85,B 0,C 180,E1 -13244.619,E2 -13244.619} C_VEL
LIN {X 0,Y 361.943,Z 348.212,A -85,B 0,C 180,E1 -13248.098,E2 -13248.098} C_VEL
LIN {X 0,Y 361.879,Z 348.223,A -85,B 0,C 180,E1 -13251.652,E2 -13251.652} C_VEL
LIN {X 0,Y 361.915,Z 348.217,A -85,B 0,C 180,E1 -13255.289,E2 -13255.289} C_VEL
LIN {X 0,Y 361.909,Z 348.217,A -85,B 0,C 180,E1 -13257.777,E2 -13257.777} C_VEL
LIN {X 0,Y 361.833,Z 348.229,A -85,B 0,C 180,E1 -13261.285,E2 -13261.285} C_VEL
LIN {X 0,Y 361.839,Z 348.223,A -85,B 0,C 180,E1 -13264.299,E2 -13264.299} C_VEL
LIN {X 0,Y 361.861,Z 348.225,A -85,B 0,C 180,E1 -13267.225,E2 -13267.225} C_VEL
LIN {X 0,Y 361.859,Z 348.224,A -85,B 0,C 180,E1 -13269.14,E2 -13269.14} C_VEL
LIN {X 0,Y 361.182,Z 348.305,A -85,B 0,C 180,E1 -13270.07,E2 -13270.07} C_VEL
LIN {X 0,Y 358.336,Z 348.661,A -85,B 0,C 180,E1 -13271.582,E2 -13271.582} C_VEL
LIN {X 0,Y 355.942,Z 348.961,A -85,B 0,C 180,E1 -13272.805,E2 -13272.805} C_VEL
LIN {X 0,Y 354.929,Z 349.085,A -85,B 0,C 180,E1 -13273.751,E2 -13273.751} C_VEL
LIN {X 0,Y 354.853,Z 349.093,A -85,B 0,C 180,E1 -13274.072,E2 -13274.072} C_VEL
LIN {X 0,Y 354.825,Z 349.097,A -85,B 0,C 180,E1 -13277.669,E2 -13277.669} C_VEL
LIN {X 0,Y 354.823,Z 349.1,A -85,B 0,C 180,E1 -13280.669,E2 -13280.669} C_VEL
LIN {X 0,Y 354.808,Z 349.1,A -85,B 0,C 180,E1 -13284.301,E2 -13284.301} C_VEL
LIN {X 0,Y 354.773,Z 349.103,A -85,B 0,C 180,E1 -13287.667,E2 -13287.667} C_VEL
LIN {X 0,Y 354.855,Z 349.098,A -85,B 0,C 180,E1 -13290.622,E2 -13290.622} C_VEL
LIN {X 0,Y 354.886,Z 349.091,A -85,B 0,C 180,E1 -13294.173,E2 -13294.173} C_VEL
LIN {X 0,Y 354.878,Z 349.091,A -85,B 0,C 180,E1 -13297.898,E2 -13297.898} C_VEL
LIN {X 0,Y 354.91,Z 349.088,A -85,B 0,C 180,E1 -13301.892,E2 -13301.892} C_VEL
LIN {X 0,Y 354.93,Z 349.086,A -85,B 0,C 180,E1 -13305.981,E2 -13305.981} C_VEL
LIN {X 0,Y 354.97,Z 349.08,A -85,B 0,C 180,E1 -13309.737,E2 -13309.737} C_VEL
LIN {X 0,Y 355.102,Z 349.067,A -85,B 0,C 180,E1 -13312.038,E2 -13312.038} C_VEL
LIN {X 0,Y 355.081,Z 349.068,A -85,B 0,C 180,E1 -13314.322,E2 -13314.322} C_VEL
